KUKA KRL program: MyProgram_011().src

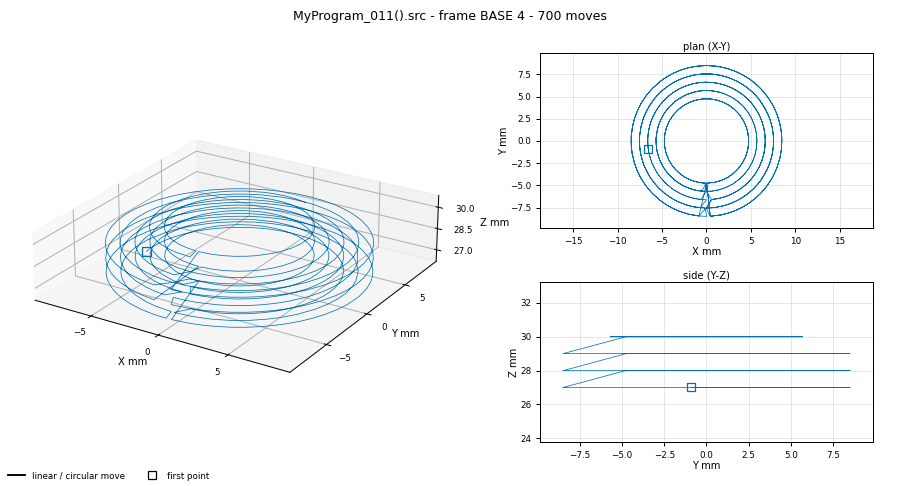
[picture p0: tool path of MyProgram_011().src in frame BASE 4, 700 of 700 moves have a stored position in this frame; points joined in program order, loops and branches not executed]
&ACCESS RVP
&REL 1
&PARAM TEMPLATE = C:\KRC\Roboter\Template\vorgabe
&PARAM EDITMASK = *
DEF MyProgram_011()
; ---- Setting reference (Base) ----
$BASE = BASE_DATA[4]

; --------------------------
; ---- Setting tool (TCP) ----
$TOOL = TOOL_DATA[3]
; --------------------------

$VEL.CP = VEL_APROX_PRINT
Startdeposition()
$VEL.CP = VEL_PRINT
LIN {X -6.5573,Y -0.8939,Z 27,A -3.0087,B 0,C 0,E1 0.1598,E2 90.0713} C_DIS
LIN {X -6.618,Y -0.1474,Z 27,A -2.9794,B 0,C 0,E1 0.1598,E2 90.0713} C_DIS
LIN {X -6.5928,Y 0.601,Z 27,A -2.9469,B 0,C 0,E1 0.1598,E2 90.0713} C_DIS
LIN {X -6.4833,Y 1.342,Z 27,A -2.9115,B 0,C 0,E1 0.1598,E2 90.0714} C_DIS
LIN {X -6.2883,Y 2.0652,Z 27,A -2.8738,B 0,C 0,E1 0.1598,E2 90.0714} C_DIS
LIN {X -6.0156,Y 2.7627,Z 27,A -2.8344,B 0,C 0,E1 0.1598,E2 90.0715} C_DIS
LIN {X -5.664,Y 3.4241,Z 27,A -2.7935,B 0,C 0,E1 0.1598,E2 90.0716} C_DIS
LIN {X -5.2401,Y 4.0414,Z 27,A -2.7519,B 0,C 0,E1 0.1598,E2 90.0717} C_DIS
LIN {X -4.7509,Y 4.6085,Z 27,A -2.7099,B 0,C 0,E1 0.1598,E2 90.0717} C_DIS
LIN {X -4.2004,Y 5.116,Z 27,A -2.6682,B 0,C 0,E1 0.1598,E2 90.0719} C_DIS
LIN {X -3.5961,Y 5.5584,Z 27,A -2.6273,B 0,C 0,E1 0.1598,E2 90.0719} C_DIS
LIN {X -2.9446,Y 5.9279,Z 27,A -2.5877,B 0,C 0,E1 0.1598,E2 90.0721} C_DIS
LIN {X -2.2557,Y 6.2218,Z 27,A -2.5499,B 0,C 0,E1 0.1598,E2 90.0721} C_DIS
LIN {X -1.5387,Y 6.4385,Z 27,A -2.5143,B 0,C 0,E1 0.1598,E2 90.0721} C_DIS
LIN {X -0.8014,Y 6.5698,Z 27,A -2.4815,B 0,C 0,E1 0.1598,E2 90.0723} C_DIS
LIN {X -0.0541,Y 6.618,Z 27,A -2.4519,B 0,C 0,E1 0.1598,E2 90.0723} C_DIS
LIN {X 0.6941,Y 6.5838,Z 27,A -2.4258,B 0,C 0,E1 0.1598,E2 90.0723} C_DIS
LIN {X 1.433,Y 6.4616,Z 27,A -2.4037,B 0,C 0,E1 0.1598,E2 90.0723} C_DIS
LIN {X 2.1541,Y 6.2595,Z 27,A -2.3856,B 0,C 0,E1 0.1598,E2 90.0723} C_DIS
LIN {X 2.8468,Y 5.9745,Z 27,A -2.3721,B 0,C 0,E1 0.1598,E2 90.0723} C_DIS
LIN {X 3.504,Y 5.6154,Z 27,A -2.3631,B 0,C 0,E1 0.1598,E2 90.0723} C_DIS
LIN {X 4.1162,Y 5.1839,Z 27,A -2.3588,B 0,C 0,E1 0.1598,E2 90.0723} C_DIS
LIN {X 4.6757,Y 4.6859,Z 27,A -2.3592,B 0,C 0,E1 0.1598,E2 90.0723} C_DIS
LIN {X 5.1746,Y 4.1272,Z 27,A -2.3645,B 0,C 0,E1 0.1598,E2 90.0723} C_DIS
LIN {X 5.6072,Y 3.5157,Z 27,A -2.3745,B 0,C 0,E1 0.1598,E2 90.0722} C_DIS
LIN {X 5.9685,Y 2.8598,Z 27,A -2.389,B 0,C 0,E1 0.1598,E2 90.0722} C_DIS
LIN {X 6.2523,Y 2.1668,Z 27,A -2.408,B 0,C 0,E1 0.1598,E2 90.0721} C_DIS
LIN {X 6.4581,Y 1.4468,Z 27,A -2.431,B 0,C 0,E1 0.1598,E2 90.0721} C_DIS
LIN {X 6.5825,Y 0.7083,Z 27,A -2.4579,B 0,C 0,E1 0.1598,E2 90.072} C_DIS
LIN {X 6.6179,Y -0.0399,Z 27,A -2.4884,B 0,C 0,E1 0.1598,E2 90.072} C_DIS
LIN {X 6.5713,Y -0.7872,Z 27,A -2.5219,B 0,C 0,E1 0.1598,E2 90.0719} C_DIS
LIN {X 6.4411,Y -1.5247,Z 27,A -2.5581,B 0,C 0,E1 0.1598,E2 90.0719} C_DIS
LIN {X 6.2271,Y -2.2424,Z 27,A -2.5965,B 0,C 0,E1 0.1598,E2 90.0719} C_DIS
LIN {X 5.9337,Y -2.9315,Z 27,A -2.6366,B 0,C 0,E1 0.1598,E2 90.0719} C_DIS
LIN {X 5.5647,Y -3.5833,Z 27,A -2.6779,B 0,C 0,E1 0.1598,E2 90.0718} C_DIS
LIN {X 5.1247,Y -4.1894,Z 27,A -2.7199,B 0,C 0,E1 0.1598,E2 90.0718} C_DIS
LIN {X 4.6171,Y -4.74,Z 27,A -2.762,B 0,C 0,E1 0.1598,E2 90.0718} C_DIS
LIN {X 4.0524,Y -5.2317,Z 27,A -2.8037,B 0,C 0,E1 0.1598,E2 90.0718} C_DIS
LIN {X 3.4359,Y -5.6569,Z 27,A -2.8444,B 0,C 0,E1 0.1598,E2 90.0717} C_DIS
LIN {X 2.7752,Y -6.0093,Z 27,A -2.8837,B 0,C 0,E1 0.1598,E2 90.0717} C_DIS
LIN {X 2.0782,Y -6.2831,Z 27,A -2.9209,B 0,C 0,E1 0.1598,E2 90.0717} C_DIS
LIN {X 1.3555,Y -6.4797,Z 27,A -2.9558,B 0,C 0,E1 0.1598,E2 90.0717} C_DIS
LIN {X 0.6148,Y -6.5905,Z 27,A -2.9877,B 0,C 0,E1 0.1598,E2 90.0716} C_DIS
LIN {X 0.6148,Y -6.5905,Z 27,A -2.9877,B 0,C 0,E1 0.1598,E2 90.0716} C_DIS
Enddeposition()
LIN {X 0.0294,Y -7.5563,Z 27,A -3.0492,B 0,C 0,E1 0.1598,E2 90.0703} C_DIS
Startdeposition()
$VEL.CP = VEL_PRINT
LIN {X 1.1276,Y -7.4726,Z 27,A -3.0064,B 0,C 0,E1 0.1598,E2 90.0715} C_DIS
LIN {X 2.4221,Y -7.16,Z 27,A -2.9457,B 0,C 0,E1 0.1598,E2 90.0716} C_DIS
LIN {X 3.4934,Y -6.6962,Z 27,A -2.8866,B 0,C 0,E1 0.1598,E2 90.0716} C_DIS
LIN {X 4.4261,Y -6.1265,Z 27,A -2.8281,B 0,C 0,E1 0.1598,E2 90.0716} C_DIS
LIN {X 5.3259,Y -5.356,Z 27,A -2.7622,B 0,C 0,E1 0.1598,E2 90.0716} C_DIS
LIN {X 5.8946,Y -4.7214,Z 27,A -2.7144,B 0,C 0,E1 0.1598,E2 90.0717} C_DIS
LIN {X 6.5048,Y -3.8483,Z 27,A -2.6545,B 0,C 0,E1 0.1598,E2 90.0716} C_DIS
LIN {X 7.0995,Y -2.5883,Z 27,A -2.5787,B 0,C 0,E1 0.1598,E2 90.0714} C_DIS
LIN {X 7.3873,Y -1.5916,Z 27,A -2.5259,B 0,C 0,E1 0.1598,E2 90.0716} C_DIS
LIN {X 7.5366,Y -0.5552,Z 27,A -2.4762,B 0,C 0,E1 0.1598,E2 90.0716} C_DIS
LIN {X 7.5438,Y 0.4481,Z 27,A -2.4333,B 0,C 0,E1 0.1598,E2 90.0717} C_DIS
LIN {X 7.425,Y 1.412,Z 27,A -2.3967,B 0,C 0,E1 0.1598,E2 90.0718} C_DIS
LIN {X 7.1966,Y 2.3052,Z 27,A -2.3672,B 0,C 0,E1 0.1598,E2 90.072} C_DIS
LIN {X 6.5668,Y 3.7404,Z 27,A -2.329,B 0,C 0,E1 0.1598,E2 90.0717} C_DIS
LIN {X 5.6905,Y 4.9679,Z 27,A -2.3091,B 0,C 0,E1 0.1598,E2 90.0717} C_DIS
LIN {X 5.2187,Y 5.4628,Z 27,A -2.3061,B 0,C 0,E1 0.1598,E2 90.0723} C_DIS
LIN {X 4.4003,Y 6.1444,Z 27,A -2.3073,B 0,C 0,E1 0.1598,E2 90.0723} C_DIS
LIN {X 3.4389,Y 6.7302,Z 27,A -2.3179,B 0,C 0,E1 0.1598,E2 90.0723} C_DIS
LIN {X 2.2888,Y 7.1954,Z 27,A -2.3408,B 0,C 0,E1 0.1598,E2 90.0723} C_DIS
LIN {X 1.4711,Y 7.4086,Z 27,A -2.362,B 0,C 0,E1 0.1598,E2 90.0723} C_DIS
LIN {X 0.6343,Y 7.527,Z 27,A -2.3879,B 0,C 0,E1 0.1598,E2 90.0723} C_DIS
LIN {X -0.2105,Y 7.5503,Z 27,A -2.4181,B 0,C 0,E1 0.1598,E2 90.0723} C_DIS
LIN {X -1.0526,Y 7.4788,Z 27,A -2.4522,B 0,C 0,E1 0.1598,E2 90.0723} C_DIS
LIN {X -2.0869,Y 7.2646,Z 27,A -2.4994,B 0,C 0,E1 0.1598,E2 90.0723} C_DIS
LIN {X -3.0794,Y 6.9019,Z 27,A -2.5514,B 0,C 0,E1 0.1598,E2 90.0721} C_DIS
LIN {X -4.0745,Y 6.365,Z 27,A -2.6107,B 0,C 0,E1 0.1598,E2 90.072} C_DIS
LIN {X -4.9827,Y 5.6816,Z 27,A -2.6729,B 0,C 0,E1 0.1598,E2 90.0718} C_DIS
LIN {X -5.5757,Y 5.0967,Z 27,A -2.7195,B 0,C 0,E1 0.1598,E2 90.0718} C_DIS
LIN {X -6.4393,Y 3.9543,Z 27,A -2.7989,B 0,C 0,E1 0.1598,E2 90.071} C_DIS
LIN {X -6.9322,Y 3.0073,Z 27,A -2.8574,B 0,C 0,E1 0.1598,E2 90.0713} C_DIS
LIN {X -7.1839,Y 2.346,Z 27,A -2.8948,B 0,C 0,E1 0.1598,E2 90.0715} C_DIS
LIN {X -7.5235,Y 0.721,Z 27,A -2.9747,B 0,C 0,E1 0.1598,E2 90.0703} C_DIS
LIN {X -7.5464,Y -0.4096,Z 27,A -3.0239,B 0,C 0,E1 0.1598,E2 90.0708} C_DIS
LIN {X -7.4299,Y -1.359,Z 27,A -3.06,B 0,C 0,E1 0.1598,E2 90.0711} C_DIS
LIN {X -7.2544,Y -2.1037,Z 27,A -3.0851,B 0,C 0,E1 0.1598,E2 90.0711} C_DIS
LIN {X -7.0048,Y -2.8269,Z 27,A -3.1065,B 0,C 0,E1 0.1598,E2 90.0711} C_DIS
LIN {X -6.5265,Y -3.8128,Z 27,A -3.1304,B 0,C 0,E1 0.1598,E2 90.0709} C_DIS
LIN {X -5.9309,Y -4.6747,Z 27,A -3.1451,B 0,C 0,E1 0.1598,E2 90.071} C_DIS
LIN {X -5.3766,Y -5.3032,Z 27,A -3.1515,B 0,C 0,E1 0.1598,E2 90.0712} C_DIS
LIN {X -4.7558,Y -5.8663,Z 27,A -3.1526,B 0,C 0,E1 0.1598,E2 90.0712} C_DIS
LIN {X -4.0775,Y -6.3584,Z 27,A -3.1486,B 0,C 0,E1 0.1598,E2 90.0712} C_DIS
LIN {X -3.3478,Y -6.7707,Z 27,A -3.1393,B 0,C 0,E1 0.1598,E2 90.0712} C_DIS
LIN {X -2.2931,Y -7.2004,Z 27,A -3.1188,B 0,C 0,E1 0.1598,E2 90.0713} C_DIS
LIN {X -1.43,Y -7.4212,Z 27,A -3.0966,B 0,C 0,E1 0.1598,E2 90.0714} C_DIS
LIN {X -0.2037,Y -7.5502,Z 27,A -3.0572,B 0,C 0,E1 0.1598,E2 90.0714} C_DIS
LIN {X -0.2037,Y -7.5502,Z 27,A -3.0572,B 0,C 0,E1 0.1598,E2 90.0714} C_DIS
Enddeposition()
LIN {X 0.0544,Y -8.4909,Z 27,A -3.0867,B 0,C 0,E1 0.1598,E2 90.0703} C_DIS
Startdeposition()
$VEL.CP = VEL_PRINT
LIN {X -0.8407,Y -8.4495,Z 27,A -3.1189,B 0,C 0,E1 0.1598,E2 90.0714} C_DIS
LIN {X -1.969,Y -8.2606,Z 27,A -3.1522,B 0,C 0,E1 0.1598,E2 90.0714} C_DIS
LIN {X -3.1017,Y -7.9005,Z 27,A -3.1784,B 0,C 0,E1 0.1598,E2 90.0712} C_DIS
LIN {X -3.874,Y -7.5517,Z 27,A -3.1919,B 0,C 0,E1 0.1598,E2 90.0712} C_DIS
LIN {X -4.6077,Y -7.1278,Z 27,A -3.2009,B 0,C 0,E1 0.1598,E2 90.0712} C_DIS
LIN {X -5.2957,Y -6.6329,Z 27,A -3.2051,B 0,C 0,E1 0.1598,E2 90.0712} C_DIS
LIN {X -6.1478,Y -5.8553,Z 27,A -3.2033,B 0,C 0,E1 0.1598,E2 90.071} C_DIS
LIN {X -6.812,Y -5.0692,Z 27,A -3.1944,B 0,C 0,E1 0.1598,E2 90.071} C_DIS
LIN {X -7.4625,Y -4.0464,Z 27,A -3.1748,B 0,C 0,E1 0.1598,E2 90.0708} C_DIS
LIN {X -7.8292,Y -3.2813,Z 27,A -3.1562,B 0,C 0,E1 0.1598,E2 90.071} C_DIS
LIN {X -8.1175,Y -2.4834,Z 27,A -3.133,B 0,C 0,E1 0.1598,E2 90.071} C_DIS
LIN {X -8.3794,Y -1.3682,Z 27,A -3.0953,B 0,C 0,E1 0.1598,E2 90.0709} C_DIS
LIN {X -8.4868,Y -0.2009,Z 27,A -3.0498,B 0,C 0,E1 0.1598,E2 90.0707} C_DIS
LIN {X -8.4719,Y 0.5615,Z 27,A -3.0174,B 0,C 0,E1 0.1598,E2 90.0711} C_DIS
LIN {X -8.2931,Y 1.8104,Z 27,A -2.9578,B 0,C 0,E1 0.1598,E2 90.0708} C_DIS
LIN {X -8.1092,Y 2.5151,Z 27,A -2.9218,B 0,C 0,E1 0.1598,E2 90.0713} C_DIS
LIN {X -7.7311,Y 3.502,Z 27,A -2.8661,B 0,C 0,E1 0.1598,E2 90.0713} C_DIS
LIN {X -7.3443,Y 4.2539,Z 27,A -2.8203,B 0,C 0,E1 0.1598,E2 90.0715} C_DIS
LIN {X -6.7611,Y 5.1353,Z 27,A -2.7615,B 0,C 0,E1 0.1598,E2 90.0715} C_DIS
LIN {X -6.0622,Y 5.9455,Z 27,A -2.7017,B 0,C 0,E1 0.1598,E2 90.0716} C_DIS
LIN {X -5.1243,Y 6.7675,Z 27,A -2.6324,B 0,C 0,E1 0.1598,E2 90.0717} C_DIS
LIN {X -4.4243,Y 7.245,Z 27,A -2.5866,B 0,C 0,E1 0.1598,E2 90.072} C_DIS
LIN {X -3.6802,Y 7.6502,Z 27,A -2.5421,B 0,C 0,E1 0.1598,E2 90.0721} C_DIS
LIN {X -2.8993,Y 7.9789,Z 27,A -2.4994,B 0,C 0,E1 0.1598,E2 90.0721} C_DIS
LIN {X -2.0894,Y 8.2279,Z 27,A -2.459,B 0,C 0,E1 0.1598,E2 90.0723} C_DIS
LIN {X -1.2587,Y 8.3946,Z 27,A -2.4213,B 0,C 0,E1 0.1598,E2 90.0723} C_DIS
LIN {X -0.0535,Y 8.4915,Z 27,A -2.3727,B 0,C 0,E1 0.1598,E2 90.0724} C_DIS
LIN {X 1.2628,Y 8.3964,Z 27,A -2.3281,B 0,C 0,E1 0.1598,E2 90.0724} C_DIS
LIN {X 2.4556,Y 8.1256,Z 27,A -2.2955,B 0,C 0,E1 0.1598,E2 90.0724} C_DIS
LIN {X 3.2184,Y 7.8542,Z 27,A -2.2788,B 0,C 0,E1 0.1598,E2 90.0724} C_DIS
LIN {X 3.9514,Y 7.5104,Z 27,A -2.2663,B 0,C 0,E1 0.1598,E2 90.0724} C_DIS
LIN {X 4.6492,Y 7.0998,Z 27,A -2.2579,B 0,C 0,E1 0.1598,E2 90.0724} C_DIS
LIN {X 5.3052,Y 6.6251,Z 27,A -2.2538,B 0,C 0,E1 0.1598,E2 90.0724} C_DIS
LIN {X 6.132,Y 5.8719,Z 27,A -2.2551,B 0,C 0,E1 0.1598,E2 90.0722} C_DIS
LIN {X 6.8769,Y 4.9736,Z 27,A -2.2656,B 0,C 0,E1 0.1598,E2 90.072} C_DIS
LIN {X 7.3469,Y 4.248,Z 27,A -2.2793,B 0,C 0,E1 0.1598,E2 90.0722} C_DIS
LIN {X 7.7408,Y 3.4783,Z 27,A -2.2975,B 0,C 0,E1 0.1598,E2 90.0722} C_DIS
LIN {X 8.0543,Y 2.6727,Z 27,A -2.3202,B 0,C 0,E1 0.1598,E2 90.0721} C_DIS
LIN {X 8.3335,Y 1.6286,Z 27,A -2.354,B 0,C 0,E1 0.1598,E2 90.0717} C_DIS
LIN {X 8.4815,Y 0.4189,Z 27,A -2.4,B 0,C 0,E1 0.1598,E2 90.0715} C_DIS
LIN {X 8.4392,Y -0.9319,Z 27,A -2.4589,B 0,C 0,E1 0.1598,E2 90.0714} C_DIS
LIN {X 8.2865,Y -1.8528,Z 27,A -2.5042,B 0,C 0,E1 0.1598,E2 90.0718} C_DIS
LIN {X 7.9336,Y -3.0156,Z 27,A -2.5665,B 0,C 0,E1 0.1598,E2 90.0714} C_DIS
LIN {X 7.5889,Y -3.7991,Z 27,A -2.6129,B 0,C 0,E1 0.1598,E2 90.0717} C_DIS
LIN {X 7.1674,Y -4.544,Z 27,A -2.6602,B 0,C 0,E1 0.1598,E2 90.0717} C_DIS
LIN {X 6.6729,Y -5.2426,Z 27,A -2.7081,B 0,C 0,E1 0.1598,E2 90.0717} C_DIS
LIN {X 6.1112,Y -5.8884,Z 27,A -2.7563,B 0,C 0,E1 0.1598,E2 90.0717} C_DIS
LIN {X 5.4874,Y -6.4744,Z 27,A -2.8041,B 0,C 0,E1 0.1598,E2 90.0717} C_DIS
LIN {X 4.8078,Y -6.9947,Z 27,A -2.8513,B 0,C 0,E1 0.1598,E2 90.0717} C_DIS
LIN {X 4.0792,Y -7.4439,Z 27,A -2.8971,B 0,C 0,E1 0.1598,E2 90.0717} C_DIS
LIN {X 3.3089,Y -7.8171,Z 27,A -2.9413,B 0,C 0,E1 0.1598,E2 90.0716} C_DIS
LIN {X 2.5048,Y -8.1107,Z 27,A -2.9833,B 0,C 0,E1 0.1598,E2 90.0716} C_DIS
LIN {X 1.6752,Y -8.3215,Z 27,A -3.0226,B 0,C 0,E1 0.1598,E2 90.0716} C_DIS
LIN {X 0.4289,Y -8.4809,Z 27,A -3.0751,B 0,C 0,E1 0.1598,E2 90.0715} C_DIS
LIN {X 0.4289,Y -8.4809,Z 27,A -3.0751,B 0,C 0,E1 0.1598,E2 90.0715} C_DIS
Enddeposition()
LIN {X 0.0007,Y -4.757,Z 28,A -2.9177,B 0,C 0,E1 0.1598,E2 90.0604} C_DIS
Startdeposition()
$VEL.CP = VEL_PRINT
LIN {X 0.0007,Y -4.757,Z 28,A -2.9234,B 0,C 0,E1 0.1598,E2 90.0661} C_DIS
LIN {X 0.963,Y -4.6517,Z 28,A -2.8885,B 0,C 0,E1 0.1598,E2 90.071} C_DIS
LIN {X 1.706,Y -4.4332,Z 28,A -2.8526,B 0,C 0,E1 0.1598,E2 90.0717} C_DIS
LIN {X 2.4029,Y -4.0959,Z 28,A -2.8127,B 0,C 0,E1 0.1598,E2 90.0717} C_DIS
LIN {X 3.0367,Y -3.6513,Z 28,A -2.7704,B 0,C 0,E1 0.1598,E2 90.0717} C_DIS
LIN {X 3.5915,Y -3.1111,Z 28,A -2.727,B 0,C 0,E1 0.1598,E2 90.0717} C_DIS
LIN {X 4.049,Y -2.4861,Z 28,A -2.6836,B 0,C 0,E1 0.1598,E2 90.0717} C_DIS
LIN {X 4.3992,Y -1.7952,Z 28,A -2.6413,B 0,C 0,E1 0.1598,E2 90.0717} C_DIS
LIN {X 4.6513,Y -0.9615,Z 28,A -2.5964,B 0,C 0,E1 0.1598,E2 90.0717} C_DIS
LIN {X 4.7407,Y -0.2897,Z 28,A -2.5647,B 0,C 0,E1 0.1598,E2 90.0719} C_DIS
LIN {X 4.7242,Y 0.4842,Z 28,A -2.5324,B 0,C 0,E1 0.1598,E2 90.0719} C_DIS
LIN {X 4.6298,Y 1.0574,Z 28,A -2.5116,B 0,C 0,E1 0.1598,E2 90.0719} C_DIS
LIN {X 4.3962,Y 1.7954,Z 28,A -2.4888,B 0,C 0,E1 0.1598,E2 90.0719} C_DIS
LIN {X 4.0466,Y 2.4862,Z 28,A -2.4723,B 0,C 0,E1 0.1598,E2 90.0719} C_DIS
LIN {X 3.5881,Y 3.1099,Z 28,A -2.4628,B 0,C 0,E1 0.1598,E2 90.0721} C_DIS
LIN {X 3.0356,Y 3.6523,Z 28,A -2.4602,B 0,C 0,E1 0.1598,E2 90.0721} C_DIS
LIN {X 2.4016,Y 4.0966,Z 28,A -2.4647,B 0,C 0,E1 0.1598,E2 90.0721} C_DIS
LIN {X 1.8838,Y 4.3598,Z 28,A -2.4727,B 0,C 0,E1 0.1598,E2 90.0722} C_DIS
LIN {X 1.1502,Y 4.6074,Z 28,A -2.4893,B 0,C 0,E1 0.1598,E2 90.0722} C_DIS
LIN {X 0.3864,Y 4.7336,Z 28,A -2.5121,B 0,C 0,E1 0.1598,E2 90.0722} C_DIS
LIN {X -0.3879,Y 4.7339,Z 28,A -2.5407,B 0,C 0,E1 0.1598,E2 90.0722} C_DIS
LIN {X -1.1516,Y 4.607,Z 28,A -2.5742,B 0,C 0,E1 0.1598,E2 90.0722} C_DIS
LIN {X -1.8851,Y 4.3592,Z 28,A -2.6117,B 0,C 0,E1 0.1598,E2 90.0721} C_DIS
LIN {X -2.5682,Y 3.9948,Z 28,A -2.6522,B 0,C 0,E1 0.1598,E2 90.072} C_DIS
LIN {X -3.1841,Y 3.5255,Z 28,A -2.6947,B 0,C 0,E1 0.1598,E2 90.0719} C_DIS
LIN {X -3.7154,Y 2.9617,Z 28,A -2.7381,B 0,C 0,E1 0.1598,E2 90.0718} C_DIS
LIN {X -4.1464,Y 2.3182,Z 28,A -2.7811,B 0,C 0,E1 0.1598,E2 90.0717} C_DIS
LIN {X -4.4674,Y 1.6136,Z 28,A -2.8227,B 0,C 0,E1 0.1598,E2 90.0716} C_DIS
LIN {X -4.6724,Y 0.8667,Z 28,A -2.8617,B 0,C 0,E1 0.1598,E2 90.0715} C_DIS
LIN {X -4.7506,Y 0.0961,Z 28,A -2.8972,B 0,C 0,E1 0.1598,E2 90.0714} C_DIS
LIN {X -4.7017,Y -0.6768,Z 28,A -2.928,B 0,C 0,E1 0.1598,E2 90.0714} C_DIS
LIN {X -4.5299,Y -1.4319,Z 28,A -2.9537,B 0,C 0,E1 0.1598,E2 90.0714} C_DIS
LIN {X -4.2369,Y -2.1487,Z 28,A -2.9733,B 0,C 0,E1 0.1598,E2 90.0714} C_DIS
LIN {X -3.8305,Y -2.8078,Z 28,A -2.9863,B 0,C 0,E1 0.1598,E2 90.0714} C_DIS
LIN {X -3.323,Y -3.3926,Z 28,A -2.9924,B 0,C 0,E1 0.1598,E2 90.0714} C_DIS
LIN {X -2.7279,Y -3.8877,Z 28,A -2.9916,B 0,C 0,E1 0.1598,E2 90.0714} C_DIS
LIN {X -2.0599,Y -4.2793,Z 28,A -2.9837,B 0,C 0,E1 0.1598,E2 90.0715} C_DIS
LIN {X -1.3374,Y -4.5575,Z 28,A -2.969,B 0,C 0,E1 0.1598,E2 90.0715} C_DIS
LIN {X -0.5793,Y -4.7151,Z 28,A -2.9479,B 0,C 0,E1 0.1598,E2 90.0716} C_DIS
LIN {X 0.0007,Y -4.757,Z 28,A -2.9284,B 0,C 0,E1 0.1598,E2 90.0716} C_DIS
Enddeposition()
LIN {X 0.0007,Y -4.757,Z 28,A -2.9284,B 0,C 0,E1 0.1598,E2 90.0716} C_DIS
Startdeposition()
$VEL.CP = VEL_PRINT
LIN {X -0.5455,Y -5.6575,Z 28,A -2.9862,B 0,C 0,E1 0.1598,E2 90.071} C_DIS
LIN {X -1.4457,Y -5.5027,Z 28,A -3.0132,B 0,C 0,E1 0.1598,E2 90.0715} C_DIS
LIN {X -2.5876,Y -5.0681,Z 28,A -3.0366,B 0,C 0,E1 0.1598,E2 90.0714} C_DIS
LIN {X -3.4004,Y -4.5542,Z 28,A -3.0447,B 0,C 0,E1 0.1598,E2 90.0714} C_DIS
LIN {X -3.9832,Y -4.0522,Z 28,A -3.0447,B 0,C 0,E1 0.1598,E2 90.0714} C_DIS
LIN {X -4.4942,Y -3.4775,Z 28,A -3.0392,B 0,C 0,E1 0.1598,E2 90.0714} C_DIS
LIN {X -4.9245,Y -2.8399,Z 28,A -3.028,B 0,C 0,E1 0.1598,E2 90.0714} C_DIS
LIN {X -5.2643,Y -2.1496,Z 28,A -3.0112,B 0,C 0,E1 0.1598,E2 90.0714} C_DIS
LIN {X -5.5044,Y -1.4186,Z 28,A -2.9891,B 0,C 0,E1 0.1598,E2 90.0714} C_DIS
LIN {X -5.6444,Y -0.6623,Z 28,A -2.9623,B 0,C 0,E1 0.1598,E2 90.0714} C_DIS
LIN {X -5.6825,Y 0.2984,Z 28,A -2.9228,B 0,C 0,E1 0.1598,E2 90.0711} C_DIS
LIN {X -5.4173,Y 1.7389,Z 28,A -2.8517,B 0,C 0,E1 0.1598,E2 90.0707} C_DIS
LIN {X -5.052,Y 2.6035,Z 28,A -2.8023,B 0,C 0,E1 0.1598,E2 90.0714} C_DIS
LIN {X -4.6641,Y 3.2461,Z 28,A -2.7611,B 0,C 0,E1 0.1598,E2 90.0717} C_DIS
LIN {X -4.1969,Y 3.8336,Z 28,A -2.7191,B 0,C 0,E1 0.1598,E2 90.0717} C_DIS
LIN {X -3.5124,Y 4.4758,Z 28,A -2.6667,B 0,C 0,E1 0.1598,E2 90.0717} C_DIS
LIN {X -2.2637,Y 5.2198,Z 28,A -2.5891,B 0,C 0,E1 0.1598,E2 90.0719} C_DIS
LIN {X -0.7561,Y 5.64,Z 28,A -2.5159,B 0,C 0,E1 0.1598,E2 90.0721} C_DIS
LIN {X 0.399,Y 5.6757,Z 28,A -2.4719,B 0,C 0,E1 0.1598,E2 90.0723} C_DIS
LIN {X 1.5931,Y 5.463,Z 28,A -2.4368,B 0,C 0,E1 0.1598,E2 90.0723} C_DIS
LIN {X 2.1802,Y 5.2494,Z 28,A -2.4242,B 0,C 0,E1 0.1598,E2 90.0723} C_DIS
LIN {X 2.9234,Y 4.8747,Z 28,A -2.4127,B 0,C 0,E1 0.1598,E2 90.0723} C_DIS
LIN {X 3.6043,Y 4.396,Z 28,A -2.4078,B 0,C 0,E1 0.1598,E2 90.0723} C_DIS
LIN {X 4.2072,Y 3.8224,Z 28,A -2.4099,B 0,C 0,E1 0.1598,E2 90.0722} C_DIS
LIN {X 4.7201,Y 3.167,Z 28,A -2.4188,B 0,C 0,E1 0.1598,E2 90.0721} C_DIS
LIN {X 5.1314,Y 2.4435,Z 28,A -2.4343,B 0,C 0,E1 0.1598,E2 90.0721} C_DIS
LIN {X 5.4343,Y 1.6684,Z 28,A -2.456,B 0,C 0,E1 0.1598,E2 90.0719} C_DIS
LIN {X 5.6202,Y 0.8572,Z 28,A -2.4837,B 0,C 0,E1 0.1598,E2 90.0719} C_DIS
LIN {X 5.6861,Y 0.0275,Z 28,A -2.5165,B 0,C 0,E1 0.1598,E2 90.0719} C_DIS
LIN {X 5.6288,Y -0.803,Z 28,A -2.5539,B 0,C 0,E1 0.1598,E2 90.0718} C_DIS
LIN {X 5.4504,Y -1.616,Z 28,A -2.5951,B 0,C 0,E1 0.1598,E2 90.0718} C_DIS
LIN {X 5.1549,Y -2.394,Z 28,A -2.6391,B 0,C 0,E1 0.1598,E2 90.0718} C_DIS
LIN {X 4.7488,Y -3.1201,Z 28,A -2.6849,B 0,C 0,E1 0.1598,E2 90.0718} C_DIS
LIN {X 4.242,Y -3.7799,Z 28,A -2.7317,B 0,C 0,E1 0.1598,E2 90.0718} C_DIS
LIN {X 3.645,Y -4.3593,Z 28,A -2.7783,B 0,C 0,E1 0.1598,E2 90.0718} C_DIS
LIN {X 2.9696,Y -4.845,Z 28,A -2.8238,B 0,C 0,E1 0.1598,E2 90.0717} C_DIS
LIN {X 2.2302,Y -5.2264,Z 28,A -2.8672,B 0,C 0,E1 0.1598,E2 90.0717} C_DIS
LIN {X 1.4431,Y -5.4959,Z 28,A -2.9075,B 0,C 0,E1 0.1598,E2 90.0717} C_DIS
LIN {X 0.6252,Y -5.648,Z 28,A -2.944,B 0,C 0,E1 0.1598,E2 90.0717} C_DIS
LIN {X 0.002,Y -5.6862,Z 28,A -2.9685,B 0,C 0,E1 0.1598,E2 90.0717} C_DIS
Enddeposition()
LIN {X 0.002,Y -5.6862,Z 28,A -2.9685,B 0,C 0,E1 0.1598,E2 90.0717} C_DIS
Startdeposition()
$VEL.CP = VEL_PRINT
LIN {X 0.5678,Y -6.5933,Z 28,A -2.9859,B 0,C 0,E1 0.1598,E2 90.071} C_DIS
LIN {X 1.325,Y -6.4863,Z 28,A -2.9541,B 0,C 0,E1 0.1598,E2 90.0716} C_DIS
LIN {X 2.0641,Y -6.2903,Z 28,A -2.9187,B 0,C 0,E1 0.1598,E2 90.0716} C_DIS
LIN {X 2.7755,Y -6.0094,Z 28,A -2.8806,B 0,C 0,E1 0.1598,E2 90.0716} C_DIS
LIN {X 3.4496,Y -5.6484,Z 28,A -2.8405,B 0,C 0,E1 0.1598,E2 90.0717} C_DIS
LIN {X 4.0795,Y -5.2147,Z 28,A -2.7989,B 0,C 0,E1 0.1598,E2 90.0717} C_DIS
LIN {X 4.653,Y -4.7087,Z 28,A -2.7563,B 0,C 0,E1 0.1598,E2 90.0717} C_DIS
LIN {X 5.1645,Y -4.1402,Z 28,A -2.7133,B 0,C 0,E1 0.1598,E2 90.0717} C_DIS
LIN {X 5.6083,Y -3.5172,Z 28,A -2.6704,B 0,C 0,E1 0.1598,E2 90.0718} C_DIS
LIN {X 5.9776,Y -2.8477,Z 28,A -2.6283,B 0,C 0,E1 0.1598,E2 90.0718} C_DIS
LIN {X 6.2652,Y -2.1391,Z 28,A -2.5875,B 0,C 0,E1 0.1598,E2 90.0718} C_DIS
LIN {X 6.4688,Y -1.4022,Z 28,A -2.5487,B 0,C 0,E1 0.1598,E2 90.0718} C_DIS
LIN {X 6.5866,Y -0.6466,Z 28,A -2.5122,B 0,C 0,E1 0.1598,E2 90.0719} C_DIS
LIN {X 6.6167,Y 0.1172,Z 28,A -2.4785,B 0,C 0,E1 0.1598,E2 90.0719} C_DIS
LIN {X 6.5616,Y 0.88,Z 28,A -2.4481,B 0,C 0,E1 0.1598,E2 90.0719} C_DIS
LIN {X 6.4145,Y 1.6304,Z 28,A -2.4216,B 0,C 0,E1 0.1598,E2 90.072} C_DIS
LIN {X 6.1829,Y 2.3591,Z 28,A -2.3991,B 0,C 0,E1 0.1598,E2 90.072} C_DIS
LIN {X 5.8718,Y 3.0575,Z 28,A -2.3809,B 0,C 0,E1 0.1598,E2 90.0721} C_DIS
LIN {X 5.4808,Y 3.7146,Z 28,A -2.3674,B 0,C 0,E1 0.1598,E2 90.0721} C_DIS
LIN {X 5.0165,Y 4.3223,Z 28,A -2.3588,B 0,C 0,E1 0.1598,E2 90.0722} C_DIS
LIN {X 4.4832,Y 4.8704,Z 28,A -2.3552,B 0,C 0,E1 0.1598,E2 90.0722} C_DIS
LIN {X 3.8915,Y 5.355,Z 28,A -2.3565,B 0,C 0,E1 0.1598,E2 90.0722} C_DIS
LIN {X 2.9648,Y 5.9228,Z 28,A -2.3665,B 0,C 0,E1 0.1598,E2 90.0722} C_DIS
LIN {X 2.0894,Y 6.2821,Z 28,A -2.3837,B 0,C 0,E1 0.1598,E2 90.0723} C_DIS
LIN {X 1.3578,Y 6.4765,Z 28,A -2.4025,B 0,C 0,E1 0.1598,E2 90.0723} C_DIS
LIN {X 0.6094,Y 6.5902,Z 28,A -2.4253,B 0,C 0,E1 0.1598,E2 90.0723} C_DIS
LIN {X -0.1472,Y 6.6173,Z 28,A -2.4521,B 0,C 0,E1 0.1598,E2 90.0723} C_DIS
LIN {X -0.902,Y 6.5575,Z 28,A -2.4825,B 0,C 0,E1 0.1598,E2 90.0723} C_DIS
LIN {X -1.6446,Y 6.4101,Z 28,A -2.5161,B 0,C 0,E1 0.1598,E2 90.0723} C_DIS
LIN {X -2.3661,Y 6.1808,Z 28,A -2.5524,B 0,C 0,E1 0.1598,E2 90.0721} C_DIS
LIN {X -3.0561,Y 5.8694,Z 28,A -2.591,B 0,C 0,E1 0.1598,E2 90.0721} C_DIS
LIN {X -3.7083,Y 5.485,Z 28,A -2.6313,B 0,C 0,E1 0.1598,E2 90.072} C_DIS
LIN {X -4.31,Y 5.0253,Z 28,A -2.6728,B 0,C 0,E1 0.1598,E2 90.072} C_DIS
LIN {X -4.8551,Y 4.4999,Z 28,A -2.7151,B 0,C 0,E1 0.1598,E2 90.0718} C_DIS
LIN {X -5.3367,Y 3.9155,Z 28,A -2.7575,B 0,C 0,E1 0.1598,E2 90.0718} C_DIS
LIN {X -5.7495,Y 3.2807,Z 28,A -2.7995,B 0,C 0,E1 0.1598,E2 90.0716} C_DIS
LIN {X -6.0883,Y 2.6037,Z 28,A -2.8405,B 0,C 0,E1 0.1598,E2 90.0716} C_DIS
LIN {X -6.3434,Y 1.8907,Z 28,A -2.88,B 0,C 0,E1 0.1598,E2 90.0715} C_DIS
LIN {X -6.5164,Y 1.1537,Z 28,A -2.9174,B 0,C 0,E1 0.1598,E2 90.0715} C_DIS
LIN {X -6.6071,Y 0.4021,Z 28,A -2.9525,B 0,C 0,E1 0.1598,E2 90.0713} C_DIS
LIN {X -6.6087,Y -0.3549,Z 28,A -2.9845,B 0,C 0,E1 0.1598,E2 90.0713} C_DIS
LIN {X -6.528,Y -1.1077,Z 28,A -3.0133,B 0,C 0,E1 0.1598,E2 90.0713} C_DIS
LIN {X -6.358,Y -1.8455,Z 28,A -3.0383,B 0,C 0,E1 0.1598,E2 90.0713} C_DIS
LIN {X -6.1068,Y -2.5598,Z 28,A -3.0593,B 0,C 0,E1 0.1598,E2 90.0713} C_DIS
LIN {X -5.7739,Y -3.2398,Z 28,A -3.0758,B 0,C 0,E1 0.1598,E2 90.0713} C_DIS
LIN {X -5.3655,Y -3.8775,Z 28,A -3.0878,B 0,C 0,E1 0.1598,E2 90.0713} C_DIS
LIN {X -4.8869,Y -4.4644,Z 28,A -3.0951,B 0,C 0,E1 0.1598,E2 90.0713} C_DIS
LIN {X -4.3445,Y -4.9926,Z 28,A -3.0976,B 0,C 0,E1 0.1598,E2 90.0713} C_DIS
LIN {X -3.7454,Y -5.4555,Z 28,A -3.0952,B 0,C 0,E1 0.1598,E2 90.0713} C_DIS
LIN {X -3.0991,Y -5.8496,Z 28,A -3.0882,B 0,C 0,E1 0.1598,E2 90.0713} C_DIS
LIN {X -2.4107,Y -6.1652,Z 28,A -3.0764,B 0,C 0,E1 0.1598,E2 90.0714} C_DIS
LIN {X -1.6904,Y -6.3984,Z 28,A -3.0599,B 0,C 0,E1 0.1598,E2 90.0714} C_DIS
LIN {X -0.9489,Y -6.5516,Z 28,A -3.0392,B 0,C 0,E1 0.1598,E2 90.0715} C_DIS
LIN {X -0.0052,Y -6.6206,Z 28,A -3.0075,B 0,C 0,E1 0.1598,E2 90.0715} C_DIS
Enddeposition()
LIN {X -0.0052,Y -6.6206,Z 28,A -3.0075,B 0,C 0,E1 0.1598,E2 90.0715} C_DIS
Startdeposition()
$VEL.CP = VEL_PRINT
LIN {X -0.6833,Y -7.5227,Z 28,A -3.0703,B 0,C 0,E1 0.1598,E2 90.0709} C_DIS
LIN {X -1.43,Y -7.4212,Z 28,A -3.0939,B 0,C 0,E1 0.1598,E2 90.0714} C_DIS
LIN {X -2.2913,Y -7.201,Z 28,A -3.1162,B 0,C 0,E1 0.1598,E2 90.0714} C_DIS
LIN {X -3.3368,Y -6.7761,Z 28,A -3.1364,B 0,C 0,E1 0.1598,E2 90.0713} C_DIS
LIN {X -4.0516,Y -6.3742,Z 28,A -3.1456,B 0,C 0,E1 0.1598,E2 90.0713} C_DIS
LIN {X -4.7187,Y -5.8976,Z 28,A -3.1499,B 0,C 0,E1 0.1598,E2 90.0713} C_DIS
LIN {X -5.3306,Y -5.3517,Z 28,A -3.1492,B 0,C 0,E1 0.1598,E2 90.0713} C_DIS
LIN {X -5.8794,Y -4.7423,Z 28,A -3.1435,B 0,C 0,E1 0.1598,E2 90.0712} C_DIS
LIN {X -6.3583,Y -4.0767,Z 28,A -3.1329,B 0,C 0,E1 0.1598,E2 90.0712} C_DIS
LIN {X -6.7613,Y -3.3628,Z 28,A -3.1174,B 0,C 0,E1 0.1598,E2 90.0712} C_DIS
LIN {X -7.0887,Y -2.611,Z 28,A -3.0977,B 0,C 0,E1 0.1598,E2 90.0712} C_DIS
LIN {X -7.3295,Y -1.8272,Z 28,A -3.0734,B 0,C 0,E1 0.1598,E2 90.0712} C_DIS
LIN {X -7.484,Y -1.0219,Z 28,A -3.045,B 0,C 0,E1 0.1598,E2 90.0712} C_DIS
LIN {X -7.5549,Y 0.1757,Z 28,A -2.9967,B 0,C 0,E1 0.1598,E2 90.0709} C_DIS
LIN {X -7.3952,Y 1.5541,Z 28,A -2.9322,B 0,C 0,E1 0.1598,E2 90.0705} C_DIS
LIN {X -7.1329,Y 2.4973,Z 28,A -2.8834,B 0,C 0,E1 0.1598,E2 90.0712} C_DIS
LIN {X -6.7699,Y 3.3575,Z 28,A -2.8338,B 0,C 0,E1 0.1598,E2 90.0714} C_DIS
LIN {X -5.9032,Y 4.7191,Z 28,A -2.7438,B 0,C 0,E1 0.1598,E2 90.0709} C_DIS
LIN {X -5.2951,Y 5.3855,Z 28,A -2.694,B 0,C 0,E1 0.1598,E2 90.0717} C_DIS
LIN {X -4.757,Y 5.8666,Z 28,A -2.6539,B 0,C 0,E1 0.1598,E2 90.0719} C_DIS
LIN {X -4.1759,Y 6.2949,Z 28,A -2.6145,B 0,C 0,E1 0.1598,E2 90.0719} C_DIS
LIN {X -3.5561,Y 6.665,Z 28,A -2.576,B 0,C 0,E1 0.1598,E2 90.0721} C_DIS
LIN {X -2.5752,Y 7.1043,Z 28,A -2.5212,B 0,C 0,E1 0.1598,E2 90.0721} C_DIS
LIN {X -1.4796,Y 7.407,Z 28,A -2.468,B 0,C 0,E1 0.1598,E2 90.0722} C_DIS
LIN {X -0.4661,Y 7.5426,Z 28,A -2.4249,B 0,C 0,E1 0.1598,E2 90.0723} C_DIS
LIN {X 0.7661,Y 7.5148,Z 28,A -2.3806,B 0,C 0,E1 0.1598,E2 90.0723} C_DIS
LIN {X 1.6891,Y 7.3611,Z 28,A -2.353,B 0,C 0,E1 0.1598,E2 90.0724} C_DIS
LIN {X 2.8073,Y 7.0176,Z 28,A -2.3262,B 0,C 0,E1 0.1598,E2 90.0724} C_DIS
LIN {X 4.0105,Y 6.4045,Z 28,A -2.3077,B 0,C 0,E1 0.1598,E2 90.0722} C_DIS
LIN {X 4.8373,Y 5.806,Z 28,A -2.3026,B 0,C 0,E1 0.1598,E2 90.0722} C_DIS
LIN {X 5.4597,Y 5.2216,Z 28,A -2.3045,B 0,C 0,E1 0.1598,E2 90.0723} C_DIS
LIN {X 6.0154,Y 4.5735,Z 28,A -2.3114,B 0,C 0,E1 0.1598,E2 90.0722} C_DIS
LIN {X 7.0188,Y 2.8045,Z 28,A -2.349,B 0,C 0,E1 0.1598,E2 90.0715} C_DIS
LIN {X 7.3743,Y 1.6355,Z 28,A -2.3857,B 0,C 0,E1 0.1598,E2 90.0715} C_DIS
LIN {X 7.504,Y 0.8928,Z 28,A -2.4129,B 0,C 0,E1 0.1598,E2 90.0719} C_DIS
LIN {X 7.5568,Y -0.0903,Z 28,A -2.4527,B 0,C 0,E1 0.1598,E2 90.0717} C_DIS
LIN {X 7.4782,Y -1.0928,Z 28,A -2.4983,B 0,C 0,E1 0.1598,E2 90.0717} C_DIS
LIN {X 7.2547,Y -2.1035,Z 28,A -2.5496,B 0,C 0,E1 0.1598,E2 90.0717} C_DIS
LIN {X 6.8881,Y -3.1065,Z 28,A -2.6057,B 0,C 0,E1 0.1598,E2 90.0715} C_DIS
LIN {X 6.17,Y -4.3555,Z 28,A -2.6851,B 0,C 0,E1 0.1598,E2 90.0713} C_DIS
LIN {X 5.6687,Y -4.9892,Z 28,A -2.731,B 0,C 0,E1 0.1598,E2 90.0717} C_DIS
LIN {X 5.1048,Y -5.5679,Z 28,A -2.7764,B 0,C 0,E1 0.1598,E2 90.0717} C_DIS
LIN {X 4.4805,Y -6.081,Z 28,A -2.8212,B 0,C 0,E1 0.1598,E2 90.0717} C_DIS
LIN {X 3.8048,Y -6.524,Z 28,A -2.8648,B 0,C 0,E1 0.1598,E2 90.0717} C_DIS
LIN {X 2.9021,Y -6.9773,Z 28,A -2.9172,B 0,C 0,E1 0.1598,E2 90.0716} C_DIS
LIN {X 1.6187,Y -7.3816,Z 28,A -2.9815,B 0,C 0,E1 0.1598,E2 90.0716} C_DIS
LIN {X 0.5862,Y -7.5345,Z 28,A -3.0259,B 0,C 0,E1 0.1598,E2 90.0716} C_DIS
LIN {X -0.0287,Y -7.5545,Z 28,A -3.0493,B 0,C 0,E1 0.1598,E2 90.0716} C_DIS
Enddeposition()
LIN {X -0.0287,Y -7.5545,Z 28,A -3.0493,B 0,C 0,E1 0.1598,E2 90.0716} C_DIS
Startdeposition()
$VEL.CP = VEL_PRINT
LIN {X 0.4292,Y -8.4808,Z 28,A -3.0715,B 0,C 0,E1 0.1598,E2 90.0709} C_DIS
LIN {X 1.6611,Y -8.3244,Z 28,A -3.0202,B 0,C 0,E1 0.1598,E2 90.0715} C_DIS
LIN {X 2.4827,Y -8.1178,Z 28,A -2.9814,B 0,C 0,E1 0.1598,E2 90.0715} C_DIS
LIN {X 3.2792,Y -7.8295,Z 28,A -2.9399,B 0,C 0,E1 0.1598,E2 90.0716} C_DIS
LIN {X 4.0434,Y -7.4642,Z 28,A -2.8963,B 0,C 0,E1 0.1598,E2 90.0716} C_DIS
LIN {X 4.767,Y -7.0237,Z 28,A -2.851,B 0,C 0,E1 0.1598,E2 90.0716} C_DIS
LIN {X 5.4431,Y -6.5133,Z 28,A -2.8044,B 0,C 0,E1 0.1598,E2 90.0717} C_DIS
LIN {X 6.0649,Y -5.938,Z 28,A -2.7571,B 0,C 0,E1 0.1598,E2 90.0717} C_DIS
LIN {X 6.6264,Y -5.3037,Z 28,A -2.7094,B 0,C 0,E1 0.1598,E2 90.0717} C_DIS
LIN {X 7.2913,Y -4.3515,Z 28,A -2.6442,B 0,C 0,E1 0.1598,E2 90.0717} C_DIS
LIN {X 7.8505,Y -3.2273,Z 28,A -2.5755,B 0,C 0,E1 0.1598,E2 90.0714} C_DIS
LIN {X 8.2285,Y -2.0926,Z 28,A -2.5132,B 0,C 0,E1 0.1598,E2 90.0715} C_DIS
LIN {X 8.4282,Y -1.0288,Z 28,A -2.4606,B 0,C 0,E1 0.1598,E2 90.0716} C_DIS
LIN {X 8.4916,Y 0.0464,Z 28,A -2.4124,B 0,C 0,E1 0.1598,E2 90.0716} C_DIS
LIN {X 8.4286,Y 1.0254,Z 28,A -2.3732,B 0,C 0,E1 0.1598,E2 90.0719} C_DIS
LIN {X 8.2241,Y 2.1097,Z 28,A -2.3344,B 0,C 0,E1 0.1598,E2 90.0719} C_DIS
LIN {X 7.892,Y 3.1225,Z 28,A -2.3036,B 0,C 0,E1 0.1598,E2 90.0719} C_DIS
LIN {X 7.5388,Y 3.8987,Z 28,A -2.2838,B 0,C 0,E1 0.1598,E2 90.0722} C_DIS
LIN {X 7.1096,Y 4.6355,Z 28,A -2.2683,B 0,C 0,E1 0.1598,E2 90.0722} C_DIS
LIN {X 6.4165,Y 5.5598,Z 28,A -2.2545,B 0,C 0,E1 0.1598,E2 90.0721} C_DIS
LIN {X 5.6064,Y 6.3725,Z 28,A -2.2499,B 0,C 0,E1 0.1598,E2 90.0721} C_DIS
LIN {X 4.9393,Y 6.902,Z 28,A -2.2522,B 0,C 0,E1 0.1598,E2 90.0724} C_DIS
LIN {X 4.2222,Y 7.3614,Z 28,A -2.2593,B 0,C 0,E1 0.1598,E2 90.0724} C_DIS
LIN {X 3.4632,Y 7.7476,Z 28,A -2.2709,B 0,C 0,E1 0.1598,E2 90.0724} C_DIS
LIN {X 2.6693,Y 8.0561,Z 28,A -2.2872,B 0,C 0,E1 0.1598,E2 90.0724} C_DIS
LIN {X 1.8485,Y 8.2832,Z 28,A -2.3079,B 0,C 0,E1 0.1598,E2 90.0724} C_DIS
LIN {X 1.0091,Y 8.4272,Z 28,A -2.3328,B 0,C 0,E1 0.1598,E2 90.0724} C_DIS
LIN {X -0.0535,Y 8.4915,Z 28,A -2.3694,B 0,C 0,E1 0.1598,E2 90.0724} C_DIS
LIN {X -1.2512,Y 8.3956,Z 28,A -2.4176,B 0,C 0,E1 0.1598,E2 90.0724} C_DIS
LIN {X -2.0826,Y 8.2295,Z 28,A -2.4554,B 0,C 0,E1 0.1598,E2 90.0723} C_DIS
LIN {X -2.8932,Y 7.981,Z 28,A -2.4958,B 0,C 0,E1 0.1598,E2 90.0723} C_DIS
LIN {X -3.6748,Y 7.6527,Z 28,A -2.5385,B 0,C 0,E1 0.1598,E2 90.0721} C_DIS
LIN {X -4.4197,Y 7.2478,Z 28,A -2.583,B 0,C 0,E1 0.1598,E2 90.0721} C_DIS
LIN {X -5.1203,Y 6.7704,Z 28,A -2.629,B 0,C 0,E1 0.1598,E2 90.072} C_DIS
LIN {X -6.0622,Y 5.9455,Z 28,A -2.6983,B 0,C 0,E1 0.1598,E2 90.0716} C_DIS
LIN {X -6.759,Y 5.138,Z 28,A -2.7581,B 0,C 0,E1 0.1598,E2 90.0716} C_DIS
LIN {X -7.3429,Y 4.2563,Z 28,A -2.8168,B 0,C 0,E1 0.1598,E2 90.0715} C_DIS
LIN {X -7.7302,Y 3.5041,Z 28,A -2.8628,B 0,C 0,E1 0.1598,E2 90.0715} C_DIS
LIN {X -8.1087,Y 2.5166,Z 28,A -2.9181,B 0,C 0,E1 0.1598,E2 90.0711} C_DIS
LIN {X -8.3768,Y 1.3752,Z 28,A -2.976,B 0,C 0,E1 0.1598,E2 90.0709} C_DIS
LIN {X -8.4719,Y 0.5625,Z 28,A -3.0139,B 0,C 0,E1 0.1598,E2 90.071} C_DIS
LIN {X -8.4654,Y -0.6204,Z 28,A -3.0633,B 0,C 0,E1 0.1598,E2 90.0707} C_DIS
LIN {X -8.3785,Y -1.3738,Z 28,A -3.0923,B 0,C 0,E1 0.1598,E2 90.071} C_DIS
LIN {X -8.1326,Y -2.4291,Z 28,A -3.1277,B 0,C 0,E1 0.1598,E2 90.0709} C_DIS
LIN {X -7.843,Y -3.2461,Z 28,A -3.1518,B 0,C 0,E1 0.1598,E2 90.071} C_DIS
LIN {X -7.4713,Y -4.0292,Z 28,A -3.1712,B 0,C 0,E1 0.1598,E2 90.071} C_DIS
LIN {X -6.8125,Y -5.0685,Z 28,A -3.1908,B 0,C 0,E1 0.1598,E2 90.0708} C_DIS
LIN {X -6.2115,Y -5.7883,Z 28,A -3.1994,B 0,C 0,E1 0.1598,E2 90.071} C_DIS
LIN {X -5.2984,Y -6.6307,Z 28,A -3.2015,B 0,C 0,E1 0.1598,E2 90.071} C_DIS
LIN {X -4.6103,Y -7.1261,Z 28,A -3.1974,B 0,C 0,E1 0.1598,E2 90.0712} C_DIS
LIN {X -3.8762,Y -7.5505,Z 28,A -3.1885,B 0,C 0,E1 0.1598,E2 90.0712} C_DIS
LIN {X -3.1035,Y -7.8997,Z 28,A -3.1751,B 0,C 0,E1 0.1598,E2 90.0712} C_DIS
LIN {X -1.9602,Y -8.2628,Z 28,A -3.1485,B 0,C 0,E1 0.1598,E2 90.0713} C_DIS
LIN {X -0.8412,Y -8.4495,Z 28,A -3.1155,B 0,C 0,E1 0.1598,E2 90.0713} C_DIS
LIN {X -0.8412,Y -8.4495,Z 28,A -3.1155,B 0,C 0,E1 0.1598,E2 90.0714} C_DIS
Enddeposition()
LIN {X 0.0007,Y -4.757,Z 29,A -2.9129,B 0,C 0,E1 0.1598,E2 90.0604} C_DIS
Startdeposition()
$VEL.CP = VEL_PRINT
LIN {X 0.0007,Y -4.757,Z 29,A -2.9186,B 0,C 0,E1 0.1598,E2 90.0661} C_DIS
LIN {X -0.6666,Y -4.7028,Z 29,A -2.9457,B 0,C 0,E1 0.1598,E2 90.071} C_DIS
LIN {X -1.3207,Y -4.5623,Z 29,A -2.9644,B 0,C 0,E1 0.1598,E2 90.0716} C_DIS
LIN {X -2.0351,Y -4.2906,Z 29,A -2.9791,B 0,C 0,E1 0.1598,E2 90.0716} C_DIS
LIN {X -2.5375,Y -4.0141,Z 29,A -2.9858,B 0,C 0,E1 0.1598,E2 90.0716} C_DIS
LIN {X -3.0035,Y -3.6798,Z 29,A -2.9888,B 0,C 0,E1 0.1598,E2 90.0716} C_DIS
LIN {X -3.5541,Y -3.1495,Z 29,A -2.9864,B 0,C 0,E1 0.1598,E2 90.0714} C_DIS
LIN {X -3.9083,Y -2.6986,Z 29,A -2.9803,B 0,C 0,E1 0.1598,E2 90.0714} C_DIS
LIN {X -4.2055,Y -2.2079,Z 29,A -2.9705,B 0,C 0,E1 0.1598,E2 90.0714} C_DIS
LIN {X -4.5041,Y -1.5044,Z 29,A -2.9516,B 0,C 0,E1 0.1598,E2 90.0714} C_DIS
LIN {X -4.6878,Y -0.7626,Z 29,A -2.9269,B 0,C 0,E1 0.1598,E2 90.0714} C_DIS
LIN {X -4.75,Y -0.0008,Z 29,A -2.897,B 0,C 0,E1 0.1598,E2 90.0714} C_DIS
LIN {X -4.6878,Y 0.761,Z 29,A -2.8625,B 0,C 0,E1 0.1598,E2 90.0714} C_DIS
LIN {X -4.5051,Y 1.5031,Z 29,A -2.8244,B 0,C 0,E1 0.1598,E2 90.0715} C_DIS
LIN {X -4.2071,Y 2.2071,Z 29,A -2.7837,B 0,C 0,E1 0.1598,E2 90.0716} C_DIS
LIN {X -3.7979,Y 2.8528,Z 29,A -2.7413,B 0,C 0,E1 0.1598,E2 90.0717} C_DIS
LIN {X -3.2906,Y 3.4246,Z 29,A -2.6985,B 0,C 0,E1 0.1598,E2 90.0718} C_DIS
LIN {X -2.6987,Y 3.9083,Z 29,A -2.6563,B 0,C 0,E1 0.1598,E2 90.0719} C_DIS
LIN {X -2.208,Y 4.2054,Z 29,A -2.6257,B 0,C 0,E1 0.1598,E2 90.072} C_DIS
LIN {X -1.5045,Y 4.5041,Z 29,A -2.5872,B 0,C 0,E1 0.1598,E2 90.072} C_DIS
LIN {X -0.9509,Y 4.6537,Z 29,A -2.5604,B 0,C 0,E1 0.1598,E2 90.0721} C_DIS
LIN {X -0.1922,Y 4.7468,Z 29,A -2.5285,B 0,C 0,E1 0.1598,E2 90.0721} C_DIS
LIN {X 0.5717,Y 4.7151,Z 29,A -2.5017,B 0,C 0,E1 0.1598,E2 90.0722} C_DIS
LIN {X 1.3209,Y 4.5633,Z 29,A -2.4805,B 0,C 0,E1 0.1598,E2 90.0722} C_DIS
LIN {X 2.0355,Y 4.2918,Z 29,A -2.4657,B 0,C 0,E1 0.1598,E2 90.0722} C_DIS
LIN {X 2.6978,Y 3.9097,Z 29,A -2.4574,B 0,C 0,E1 0.1598,E2 90.0722} C_DIS
LIN {X 3.2903,Y 3.4266,Z 29,A -2.456,B 0,C 0,E1 0.1598,E2 90.0722} C_DIS
LIN {X 3.7985,Y 2.8553,Z 29,A -2.4615,B 0,C 0,E1 0.1598,E2 90.0721} C_DIS
LIN {X 4.2061,Y 2.2082,Z 29,A -2.474,B 0,C 0,E1 0.1598,E2 90.0721} C_DIS
LIN {X 4.5045,Y 1.5045,Z 29,A -2.4928,B 0,C 0,E1 0.1598,E2 90.072} C_DIS
LIN {X 4.6537,Y 0.9508,Z 29,A -2.511,B 0,C 0,E1 0.1598,E2 90.072} C_DIS
LIN {X 4.7442,Y 0.1918,Z 29,A -2.5397,B 0,C 0,E1 0.1598,E2 90.0719} C_DIS
LIN {X 4.734,Y -0.3814,Z 29,A -2.5645,B 0,C 0,E1 0.1598,E2 90.0719} C_DIS
LIN {X 4.6116,Y -1.1359,Z 29,A -2.6011,B 0,C 0,E1 0.1598,E2 90.0718} C_DIS
LIN {X 4.3699,Y -1.8611,Z 29,A -2.6408,B 0,C 0,E1 0.1598,E2 90.0718} C_DIS
LIN {X 4.0154,Y -2.5383,Z 29,A -2.6827,B 0,C 0,E1 0.1598,E2 90.0718} C_DIS
LIN {X 3.5563,Y -3.1497,Z 29,A -2.7256,B 0,C 0,E1 0.1598,E2 90.0718} C_DIS
LIN {X 3.0055,Y -3.6801,Z 29,A -2.7684,B 0,C 0,E1 0.1598,E2 90.0718} C_DIS
LIN {X 2.3765,Y -4.115,Z 29,A -2.81,B 0,C 0,E1 0.1598,E2 90.0718} C_DIS
LIN {X 1.5952,Y -4.4741,Z 29,A -2.854,B 0,C 0,E1 0.1598,E2 90.0718} C_DIS
LIN {X 0.9508,Y -4.6538,Z 29,A -2.8853,B 0,C 0,E1 0.1598,E2 90.0718} C_DIS
LIN {X 0.192,Y -4.7489,Z 29,A -2.9172,B 0,C 0,E1 0.1598,E2 90.0717} C_DIS
LIN {X 0.192,Y -4.7489,Z 29,A -2.9172,B 0,C 0,E1 0.1598,E2 90.0717} C_DIS
Enddeposition()
LIN {X -0.0133,Y -5.6862,Z 29,A -2.9635,B 0,C 0,E1 0.1598,E2 90.0705} C_DIS
Startdeposition()
$VEL.CP = VEL_PRINT
LIN {X 0.6191,Y -5.6481,Z 29,A -2.9398,B 0,C 0,E1 0.1598,E2 90.0716} C_DIS
LIN {X 1.4488,Y -5.4937,Z 29,A -2.9029,B 0,C 0,E1 0.1598,E2 90.0716} C_DIS
LIN {X 2.2472,Y -5.2194,Z 29,A -2.8619,B 0,C 0,E1 0.1598,E2 90.0717} C_DIS
LIN {X 2.9952,Y -4.8282,Z 29,A -2.8178,B 0,C 0,E1 0.1598,E2 90.0717} C_DIS
LIN {X 3.6773,Y -4.3311,Z 29,A -2.7715,B 0,C 0,E1 0.1598,E2 90.0717} C_DIS
LIN {X 4.2791,Y -3.7391,Z 29,A -2.7242,B 0,C 0,E1 0.1598,E2 90.0717} C_DIS
LIN {X 4.7856,Y -3.0637,Z 29,A -2.6768,B 0,C 0,E1 0.1598,E2 90.0717} C_DIS
LIN {X 5.1869,Y -2.3211,Z 29,A -2.6304,B 0,C 0,E1 0.1598,E2 90.0717} C_DIS
LIN {X 5.4728,Y -1.5268,Z 29,A -2.586,B 0,C 0,E1 0.1598,E2 90.0717} C_DIS
LIN {X 5.6386,Y -0.6992,Z 29,A -2.5447,B 0,C 0,E1 0.1598,E2 90.0718} C_DIS
LIN {X 5.6813,Y 0.1438,Z 29,A -2.5072,B 0,C 0,E1 0.1598,E2 90.0718} C_DIS
LIN {X 5.5992,Y 0.9842,Z 29,A -2.4745,B 0,C 0,E1 0.1598,E2 90.0718} C_DIS
LIN {X 5.3921,Y 1.803,Z 29,A -2.4473,B 0,C 0,E1 0.1598,E2 90.0719} C_DIS
LIN {X 5.0653,Y 2.5818,Z 29,A -2.4263,B 0,C 0,E1 0.1598,E2 90.0719} C_DIS
LIN {X 4.6248,Y 3.3022,Z 29,A -2.4119,B 0,C 0,E1 0.1598,E2 90.072} C_DIS
LIN {X 4.085,Y 3.9514,Z 29,A -2.4043,B 0,C 0,E1 0.1598,E2 90.0721} C_DIS
LIN {X 3.4544,Y 4.5128,Z 29,A -2.4038,B 0,C 0,E1 0.1598,E2 90.0721} C_DIS
LIN {X 2.748,Y 4.9753,Z 29,A -2.4103,B 0,C 0,E1 0.1598,E2 90.0722} C_DIS
LIN {X 1.9809,Y 5.3283,Z 29,A -2.4236,B 0,C 0,E1 0.1598,E2 90.0722} C_DIS
LIN {X 1.1698,Y 5.5633,Z 29,A -2.4436,B 0,C 0,E1 0.1598,E2 90.0722} C_DIS
LIN {X 0.3328,Y 5.675,Z 29,A -2.4698,B 0,C 0,E1 0.1598,E2 90.0722} C_DIS
LIN {X -0.5116,Y 5.6623,Z 29,A -2.5015,B 0,C 0,E1 0.1598,E2 90.0722} C_DIS
LIN {X -1.345,Y 5.5247,Z 29,A -2.538,B 0,C 0,E1 0.1598,E2 90.0722} C_DIS
LIN {X -2.106,Y 5.2868,Z 29,A -2.5761,B 0,C 0,E1 0.1598,E2 90.0721} C_DIS
LIN {X -3.0284,Y 4.811,Z 29,A -2.6302,B 0,C 0,E1 0.1598,E2 90.072} C_DIS
LIN {X -3.6969,Y 4.3187,Z 29,A -2.6756,B 0,C 0,E1 0.1598,E2 90.0719} C_DIS
LIN {X -4.2858,Y 3.7336,Z 29,A -2.722,B 0,C 0,E1 0.1598,E2 90.0718} C_DIS
LIN {X -4.7846,Y 3.0699,Z 29,A -2.7684,B 0,C 0,E1 0.1598,E2 90.0717} C_DIS
LIN {X -5.1807,Y 2.3403,Z 29,A -2.8137,B 0,C 0,E1 0.1598,E2 90.0715} C_DIS
LIN {X -5.5464,Y 1.2703,Z 29,A -2.8721,B 0,C 0,E1 0.1598,E2 90.0712} C_DIS
LIN {X -5.671,Y 0.4096,Z 29,A -2.9133,B 0,C 0,E1 0.1598,E2 90.0713} C_DIS
LIN {X -5.6783,Y -0.286,Z 29,A -2.943,B 0,C 0,E1 0.1598,E2 90.0713} C_DIS
LIN {X -5.601,Y -0.9774,Z 29,A -2.9694,B 0,C 0,E1 0.1598,E2 90.0713} C_DIS
LIN {X -5.4392,Y -1.6539,Z 29,A -2.9921,B 0,C 0,E1 0.1598,E2 90.0713} C_DIS
LIN {X -5.1971,Y -2.3061,Z 29,A -3.0108,B 0,C 0,E1 0.1598,E2 90.0713} C_DIS
LIN {X -4.875,Y -2.9226,Z 29,A -3.0251,B 0,C 0,E1 0.1598,E2 90.0713} C_DIS
LIN {X -4.2655,Y -3.7651,Z 29,A -3.0382,B 0,C 0,E1 0.1598,E2 90.0712} C_DIS
LIN {X -3.5966,Y -4.4018,Z 29,A -3.0407,B 0,C 0,E1 0.1598,E2 90.0713} C_DIS
LIN {X -2.995,Y -4.8304,Z 29,A -3.0369,B 0,C 0,E1 0.1598,E2 90.0714} C_DIS
LIN {X -2.3436,Y -5.1784,Z 29,A -3.0278,B 0,C 0,E1 0.1598,E2 90.0714} C_DIS
LIN {X -1.6525,Y -5.4394,Z 29,A -3.0135,B 0,C 0,E1 0.1598,E2 90.0715} C_DIS
LIN {X -0.9334,Y -5.609,Z 29,A -2.9944,B 0,C 0,E1 0.1598,E2 90.0715} C_DIS
LIN {X -0.0133,Y -5.6862,Z 29,A -2.9639,B 0,C 0,E1 0.1598,E2 90.0716} C_DIS
Enddeposition()
LIN {X -0.0133,Y -5.6862,Z 29,A -2.9639,B 0,C 0,E1 0.1598,E2 90.0716} C_DIS
Startdeposition()
$VEL.CP = VEL_PRINT
LIN {X -0.6208,Y -6.5907,Z 29,A -3.0242,B 0,C 0,E1 0.1598,E2 90.071} C_DIS
LIN {X -1.3808,Y -6.4718,Z 29,A -3.0475,B 0,C 0,E1 0.1598,E2 90.0715} C_DIS
LIN {X -2.1223,Y -6.2676,Z 29,A -3.0661,B 0,C 0,E1 0.1598,E2 90.0715} C_DIS
LIN {X -2.8355,Y -5.9798,Z 29,A -3.08,B 0,C 0,E1 0.1598,E2 90.0715} C_DIS
LIN {X -3.5119,Y -5.6133,Z 29,A -3.0893,B 0,C 0,E1 0.1598,E2 90.0714} C_DIS
LIN {X -4.1379,Y -5.1663,Z 29,A -3.0933,B 0,C 0,E1 0.1598,E2 90.0714} C_DIS
LIN {X -4.7092,Y -4.651,Z 29,A -3.0924,B 0,C 0,E1 0.1598,E2 90.0714} C_DIS
LIN {X -5.2165,Y -4.0727,Z 29,A -3.0865,B 0,C 0,E1 0.1598,E2 90.0713} C_DIS
LIN {X -5.6539,Y -3.44,Z 29,A -3.0757,B 0,C 0,E1 0.1598,E2 90.0713} C_DIS
LIN {X -6.0146,Y -2.7607,Z 29,A -3.0602,B 0,C 0,E1 0.1598,E2 90.0713} C_DIS
LIN {X -6.2939,Y -2.0441,Z 29,A -3.0401,B 0,C 0,E1 0.1598,E2 90.0713} C_DIS
LIN {X -6.4899,Y -1.3003,Z 29,A -3.0159,B 0,C 0,E1 0.1598,E2 90.0713} C_DIS
LIN {X -6.5981,Y -0.5386,Z 29,A -2.9877,B 0,C 0,E1 0.1598,E2 90.0713} C_DIS
LIN {X -6.6161,Y 0.2303,Z 29,A -2.9558,B 0,C 0,E1 0.1598,E2 90.0713} C_DIS
LIN {X -6.5446,Y 0.9964,Z 29,A -2.9209,B 0,C 0,E1 0.1598,E2 90.0713} C_DIS
LIN {X -6.3856,Y 1.749,Z 29,A -2.8832,B 0,C 0,E1 0.1598,E2 90.0714} C_DIS
LIN {X -6.1392,Y 2.4777,Z 29,A -2.8434,B 0,C 0,E1 0.1598,E2 90.0715} C_DIS
LIN {X -5.8115,Y 3.1737,Z 29,A -2.802,B 0,C 0,E1 0.1598,E2 90.0715} C_DIS
LIN {X -5.4017,Y 3.8247,Z 29,A -2.7594,B 0,C 0,E1 0.1598,E2 90.0717} C_DIS
LIN {X -4.9223,Y 4.4264,Z 29,A -2.7163,B 0,C 0,E1 0.1598,E2 90.0717} C_DIS
LIN {X -4.3747,Y 4.9668,Z 29,A -2.6734,B 0,C 0,E1 0.1598,E2 90.0719} C_DIS
LIN {X -3.7684,Y 5.4402,Z 29,A -2.631,B 0,C 0,E1 0.1598,E2 90.0719} C_DIS
LIN {X -3.112,Y 5.8414,Z 29,A -2.5899,B 0,C 0,E1 0.1598,E2 90.072} C_DIS
LIN {X -2.4136,Y 6.1638,Z 29,A -2.5505,B 0,C 0,E1 0.1598,E2 90.0721} C_DIS
LIN {X -1.6817,Y 6.4008,Z 29,A -2.5135,B 0,C 0,E1 0.1598,E2 90.0721} C_DIS
LIN {X -0.9278,Y 6.5531,Z 29,A -2.4793,B 0,C 0,E1 0.1598,E2 90.0723} C_DIS
LIN {X -0.1612,Y 6.6175,Z 29,A -2.4483,B 0,C 0,E1 0.1598,E2 90.0723} C_DIS
LIN {X 0.6075,Y 6.5896,Z 29,A -2.4211,B 0,C 0,E1 0.1598,E2 90.0723} C_DIS
LIN {X 1.3683,Y 6.4761,Z 29,A -2.3978,B 0,C 0,E1 0.1598,E2 90.0723} C_DIS
LIN {X 2.1107,Y 6.2747,Z 29,A -2.379,B 0,C 0,E1 0.1598,E2 90.0723} C_DIS
LIN {X 3.124,Y 5.8403,Z 29,A -2.3599,B 0,C 0,E1 0.1598,E2 90.0723} C_DIS
LIN {X 3.9436,Y 5.3171,Z 29,A -2.3518,B 0,C 0,E1 0.1598,E2 90.0723} C_DIS
LIN {X 4.5395,Y 4.8172,Z 29,A -2.3511,B 0,C 0,E1 0.1598,E2 90.0723} C_DIS
LIN {X 5.0729,Y 4.2511,Z 29,A -2.3554,B 0,C 0,E1 0.1598,E2 90.0723} C_DIS
LIN {X 5.5363,Y 3.6267,Z 29,A -2.3648,B 0,C 0,E1 0.1598,E2 90.0722} C_DIS
LIN {X 5.9232,Y 2.952,Z 29,A -2.3792,B 0,C 0,E1 0.1598,E2 90.0722} C_DIS
LIN {X 6.23,Y 2.2372,Z 29,A -2.3983,B 0,C 0,E1 0.1598,E2 90.0721} C_DIS
LIN {X 6.4494,Y 1.491,Z 29,A -2.4219,B 0,C 0,E1 0.1598,E2 90.0721} C_DIS
LIN {X 6.5775,Y 0.7239,Z 29,A -2.4498,B 0,C 0,E1 0.1598,E2 90.072} C_DIS
LIN {X 6.6174,Y -0.0526,Z 29,A -2.4814,B 0,C 0,E1 0.1598,E2 90.072} C_DIS
LIN {X 6.568,Y -0.8287,Z 29,A -2.5163,B 0,C 0,E1 0.1598,E2 90.0719} C_DIS
LIN {X 6.4253,Y -1.5935,Z 29,A -2.5541,B 0,C 0,E1 0.1598,E2 90.0719} C_DIS
LIN {X 6.1951,Y -2.3364,Z 29,A -2.5942,B 0,C 0,E1 0.1598,E2 90.0719} C_DIS
LIN {X 5.8775,Y -3.0464,Z 29,A -2.6361,B 0,C 0,E1 0.1598,E2 90.0718} C_DIS
LIN {X 5.4804,Y -3.7151,Z 29,A -2.6792,B 0,C 0,E1 0.1598,E2 90.0718} C_DIS
LIN {X 5.0044,Y -4.3303,Z 29,A -2.7229,B 0,C 0,E1 0.1598,E2 90.0718} C_DIS
LIN {X 4.4626,Y -4.8882,Z 29,A -2.7665,B 0,C 0,E1 0.1598,E2 90.0718} C_DIS
LIN {X 3.7011,Y -5.4927,Z 29,A -2.8202,B 0,C 0,E1 0.1598,E2 90.0716} C_DIS
LIN {X 2.7577,Y -6.0176,Z 29,A -2.8772,B 0,C 0,E1 0.1598,E2 90.0716} C_DIS
LIN {X 2.0403,Y -6.2971,Z 29,A -2.9155,B 0,C 0,E1 0.1598,E2 90.0716} C_DIS
LIN {X 1.2949,Y -6.4895,Z 29,A -2.951,B 0,C 0,E1 0.1598,E2 90.0716} C_DIS
LIN {X 0.5327,Y -6.5966,Z 29,A -2.9835,B 0,C 0,E1 0.1598,E2 90.0716} C_DIS
LIN {X 0.5327,Y -6.5966,Z 29,A -2.9835,B 0,C 0,E1 0.1598,E2 90.0716} C_DIS
Enddeposition()
LIN {X -0.0423,Y -7.5529,Z 29,A -3.0442,B 0,C 0,E1 0.1598,E2 90.0703} C_DIS
Startdeposition()
$VEL.CP = VEL_PRINT
LIN {X 0.8187,Y -7.5124,Z 29,A -3.0121,B 0,C 0,E1 0.1598,E2 90.0715} C_DIS
LIN {X 2.0741,Y -7.2685,Z 29,A -2.9557,B 0,C 0,E1 0.1598,E2 90.0716} C_DIS
LIN {X 3.0258,Y -6.9247,Z 29,A -2.9061,B 0,C 0,E1 0.1598,E2 90.0716} C_DIS
LIN {X 3.926,Y -6.4567,Z 29,A -2.8532,B 0,C 0,E1 0.1598,E2 90.0716} C_DIS
LIN {X 4.768,Y -5.8568,Z 29,A -2.7967,B 0,C 0,E1 0.1598,E2 90.0716} C_DIS
LIN {X 5.5262,Y -5.1541,Z 29,A -2.7388,B 0,C 0,E1 0.1598,E2 90.0716} C_DIS
LIN {X 6.1549,Y -4.385,Z 29,A -2.683,B 0,C 0,E1 0.1598,E2 90.0716} C_DIS
LIN {X 6.8051,Y -3.2851,Z 29,A -2.6119,B 0,C 0,E1 0.1598,E2 90.0716} C_DIS
LIN {X 7.2027,Y -2.2755,Z 29,A -2.5544,B 0,C 0,E1 0.1598,E2 90.0716} C_DIS
LIN {X 7.4151,Y -1.4338,Z 29,A -2.5108,B 0,C 0,E1 0.1598,E2 90.0718} C_DIS
LIN {X 7.5307,Y -0.5735,Z 29,A -2.4699,B 0,C 0,E1 0.1598,E2 90.0718} C_DIS
LIN {X 7.5329,Y 0.6101,Z 29,A -2.4191,B 0,C 0,E1 0.1598,E2 90.0716} C_DIS
LIN {X 7.3912,Y 1.5733,Z 29,A -2.3836,B 0,C 0,E1 0.1598,E2 90.0719} C_DIS
LIN {X 7.1087,Y 2.5633,Z 29,A -2.3518,B 0,C 0,E1 0.1598,E2 90.0719} C_DIS
LIN {X 6.7016,Y 3.4831,Z 29,A -2.3277,B 0,C 0,E1 0.1598,E2 90.072} C_DIS
LIN {X 6.2936,Y 4.1767,Z 29,A -2.3135,B 0,C 0,E1 0.1598,E2 90.0722} C_DIS
LIN {X 5.8133,Y 4.8224,Z 29,A -2.3038,B 0,C 0,E1 0.1598,E2 90.0722} C_DIS
LIN {X 5.2673,Y 5.4137,Z 29,A -2.2988,B 0,C 0,E1 0.1598,E2 90.0722} C_DIS
LIN {X 4.4116,Y 6.1366,Z 29,A -2.2996,B 0,C 0,E1 0.1598,E2 90.0722} C_DIS
LIN {X 3.4731,Y 6.7065,Z 29,A -2.3101,B 0,C 0,E1 0.1598,E2 90.0722} C_DIS
LIN {X 2.4662,Y 7.1444,Z 29,A -2.3288,B 0,C 0,E1 0.1598,E2 90.0723} C_DIS
LIN {X 1.2648,Y 7.4474,Z 29,A -2.3604,B 0,C 0,E1 0.1598,E2 90.0723} C_DIS
LIN {X 0.5221,Y 7.5389,Z 29,A -2.384,B 0,C 0,E1 0.1598,E2 90.0723} C_DIS
LIN {X -0.4709,Y 7.5423,Z 29,A -2.4205,B 0,C 0,E1 0.1598,E2 90.0723} C_DIS
LIN {X -1.4052,Y 7.4264,Z 29,A -2.4599,B 0,C 0,E1 0.1598,E2 90.0723} C_DIS
LIN {X -2.726,Y 7.0489,Z 29,A -2.5245,B 0,C 0,E1 0.1598,E2 90.0721} C_DIS
LIN {X -3.5431,Y 6.6753,Z 29,A -2.5704,B 0,C 0,E1 0.1598,E2 90.0721} C_DIS
LIN {X -4.2649,Y 6.2367,Z 29,A -2.6156,B 0,C 0,E1 0.1598,E2 90.072} C_DIS
LIN {X -5.06,Y 5.6151,Z 29,A -2.671,B 0,C 0,E1 0.1598,E2 90.0718} C_DIS
LIN {X -5.7516,Y 4.8971,Z 29,A -2.7268,B 0,C 0,E1 0.1598,E2 90.0718} C_DIS
LIN {X -6.4541,Y 3.9302,Z 29,A -2.7933,B 0,C 0,E1 0.1598,E2 90.0714} C_DIS
LIN {X -7.0526,Y 2.7159,Z 29,A -2.8663,B 0,C 0,E1 0.1598,E2 90.071} C_DIS
LIN {X -7.3858,Y 1.599,Z 29,A -2.9257,B 0,C 0,E1 0.1598,E2 90.071} C_DIS
LIN {X -7.5396,Y 0.5111,Z 29,A -2.9774,B 0,C 0,E1 0.1598,E2 90.071} C_DIS
LIN {X -7.539,Y -0.5199,Z 29,A -3.0209,B 0,C 0,E1 0.1598,E2 90.071} C_DIS
LIN {X -7.4085,Y -1.4906,Z 29,A -3.0572,B 0,C 0,E1 0.1598,E2 90.071} C_DIS
LIN {X -7.0293,Y -2.7788,Z 29,A -3.0974,B 0,C 0,E1 0.1598,E2 90.0707} C_DIS
LIN {X -6.5198,Y -3.8139,Z 29,A -3.1226,B 0,C 0,E1 0.1598,E2 90.0707} C_DIS
LIN {X -6.0535,Y -4.5163,Z 29,A -3.1355,B 0,C 0,E1 0.1598,E2 90.0711} C_DIS
LIN {X -5.5128,Y -5.1634,Z 29,A -3.1431,B 0,C 0,E1 0.1598,E2 90.0711} C_DIS
LIN {X -4.7438,Y -5.8842,Z 29,A -3.1453,B 0,C 0,E1 0.1598,E2 90.0711} C_DIS
LIN {X -3.7239,Y -6.5716,Z 29,A -3.1371,B 0,C 0,E1 0.1598,E2 90.0711} C_DIS
LIN {X -3.0328,Y -6.9217,Z 29,A -3.1267,B 0,C 0,E1 0.1598,E2 90.0713} C_DIS
LIN {X -1.7494,Y -7.3531,Z 29,A -3.098,B 0,C 0,E1 0.1598,E2 90.0713} C_DIS
LIN {X -0.7943,Y -7.5152,Z 29,A -3.0699,B 0,C 0,E1 0.1598,E2 90.0715} C_DIS
LIN {X -0.0423,Y -7.5529,Z 29,A -3.044,B 0,C 0,E1 0.1598,E2 90.0715} C_DIS
Enddeposition()
LIN {X -0.0423,Y -7.5529,Z 29,A -3.044,B 0,C 0,E1 0.1598,E2 90.0715} C_DIS
Startdeposition()
$VEL.CP = VEL_PRINT
LIN {X -0.8417,Y -8.4494,Z 29,A -3.111,B 0,C 0,E1 0.1598,E2 90.0709} C_DIS
LIN {X -2.0289,Y -8.2451,Z 29,A -3.1463,B 0,C 0,E1 0.1598,E2 90.0713} C_DIS
LIN {X -3.0371,Y -7.9238,Z 29,A -3.1697,B 0,C 0,E1 0.1598,E2 90.0713} C_DIS
LIN {X -3.8114,Y -7.5817,Z 29,A -3.1835,B 0,C 0,E1 0.1598,E2 90.0713} C_DIS
LIN {X -4.5477,Y -7.1642,Z 29,A -3.1928,B 0,C 0,E1 0.1598,E2 90.0713} C_DIS
LIN {X -5.2389,Y -6.6755,Z 29,A -3.1974,B 0,C 0,E1 0.1598,E2 90.0712} C_DIS
LIN {X -5.8781,Y -6.1205,Z 29,A -3.1974,B 0,C 0,E1 0.1598,E2 90.0712} C_DIS
LIN {X -6.4588,Y -5.5047,Z 29,A -3.1925,B 0,C 0,E1 0.1598,E2 90.0712} C_DIS
LIN {X -6.9754,Y -4.8341,Z 29,A -3.1831,B 0,C 0,E1 0.1598,E2 90.0711} C_DIS
LIN {X -7.4226,Y -4.1154,Z 29,A -3.1691,B 0,C 0,E1 0.1598,E2 90.0711} C_DIS
LIN {X -7.7957,Y -3.3556,Z 29,A -3.1506,B 0,C 0,E1 0.1598,E2 90.0711} C_DIS
LIN {X -8.0911,Y -2.5623,Z 29,A -3.1279,B 0,C 0,E1 0.1598,E2 90.0711} C_DIS
LIN {X -8.367,Y -1.4458,Z 29,A -3.0907,B 0,C 0,E1 0.1598,E2 90.0709} C_DIS
LIN {X -8.4808,Y -0.43,Z 29,A -3.0519,B 0,C 0,E1 0.1598,E2 90.0709} C_DIS
LIN {X -8.4718,Y 0.5635,Z 29,A -3.0098,B 0,C 0,E1 0.1598,E2 90.071} C_DIS
LIN {X -8.2925,Y 1.8126,Z 29,A -2.9502,B 0,C 0,E1 0.1598,E2 90.0708} C_DIS
LIN {X -8.0728,Y 2.6313,Z 29,A -2.9078,B 0,C 0,E1 0.1598,E2 90.0711} C_DIS
LIN {X -7.703,Y 3.5618,Z 29,A -2.8551,B 0,C 0,E1 0.1598,E2 90.0714} C_DIS
LIN {X -7.3336,Y 4.2727,Z 29,A -2.8116,B 0,C 0,E1 0.1598,E2 90.0716} C_DIS
LIN {X -6.7818,Y 5.1083,Z 29,A -2.7559,B 0,C 0,E1 0.1598,E2 90.0715} C_DIS
LIN {X -6.0408,Y 5.9681,Z 29,A -2.6923,B 0,C 0,E1 0.1598,E2 90.0716} C_DIS
LIN {X -5.1168,Y 6.773,Z 29,A -2.6243,B 0,C 0,E1 0.1598,E2 90.0717} C_DIS
LIN {X -4.4156,Y 7.2502,Z 29,A -2.5785,B 0,C 0,E1 0.1598,E2 90.072} C_DIS
LIN {X -3.6701,Y 7.6548,Z 29,A -2.5339,B 0,C 0,E1 0.1598,E2 90.0721} C_DIS
LIN {X -2.8879,Y 7.9827,Z 29,A -2.4912,B 0,C 0,E1 0.1598,E2 90.0721} C_DIS
LIN {X -2.0769,Y 8.2308,Z 29,A -2.4508,B 0,C 0,E1 0.1598,E2 90.0723} C_DIS
LIN {X -0.8638,Y 8.4469,Z 29,A -2.3969,B 0,C 0,E1 0.1598,E2 90.0723} C_DIS
LIN {X 0.1855,Y 8.4885,Z 29,A -2.3564,B 0,C 0,E1 0.1598,E2 90.0724} C_DIS
LIN {X 1.2708,Y 8.3951,Z 29,A -2.3202,B 0,C 0,E1 0.1598,E2 90.0724} C_DIS
LIN {X 2.2711,Y 8.182,Z 29,A -2.2923,B 0,C 0,E1 0.1598,E2 90.0724} C_DIS
LIN {X 3.2716,Y 7.8332,Z 29,A -2.2701,B 0,C 0,E1 0.1598,E2 90.0724} C_DIS
LIN {X 4.0364,Y 7.4678,Z 29,A -2.2574,B 0,C 0,E1 0.1598,E2 90.0724} C_DIS
LIN {X 5.0248,Y 6.8459,Z 29,A -2.2471,B 0,C 0,E1 0.1598,E2 90.0724} C_DIS
LIN {X 5.9377,Y 6.0653,Z 29,A -2.2464,B 0,C 0,E1 0.1598,E2 90.0722} C_DIS
LIN {X 6.5136,Y 5.4427,Z 29,A -2.2518,B 0,C 0,E1 0.1598,E2 90.0723} C_DIS
LIN {X 7.0245,Y 4.7658,Z 29,A -2.2617,B 0,C 0,E1 0.1598,E2 90.0723} C_DIS
LIN {X 7.4653,Y 4.0412,Z 29,A -2.2762,B 0,C 0,E1 0.1598,E2 90.0723} C_DIS
LIN {X 7.9133,Y 3.0805,Z 29,A -2.3003,B 0,C 0,E1 0.1598,E2 90.0719} C_DIS
LIN {X 8.2304,Y 2.0686,Z 29,A -2.3317,B 0,C 0,E1 0.1598,E2 90.0719} C_DIS
LIN {X 8.4295,Y 1.0172,Z 29,A -2.3691,B 0,C 0,E1 0.1598,E2 90.0717} C_DIS
LIN {X 8.4913,Y 0.0632,Z 29,A -2.4075,B 0,C 0,E1 0.1598,E2 90.0717} C_DIS
LIN {X 8.4404,Y -0.9216,Z 29,A -2.4513,B 0,C 0,E1 0.1598,E2 90.0717} C_DIS
LIN {X 8.2844,Y -1.8629,Z 29,A -2.4972,B 0,C 0,E1 0.1598,E2 90.0717} C_DIS
LIN {X 7.9358,Y -3.0191,Z 29,A -2.5591,B 0,C 0,E1 0.1598,E2 90.0714} C_DIS
LIN {X 7.3817,Y -4.196,Z 29,A -2.6296,B 0,C 0,E1 0.1598,E2 90.0714} C_DIS
LIN {X 6.7565,Y -5.1412,Z 29,A -2.6931,B 0,C 0,E1 0.1598,E2 90.0715} C_DIS
LIN {X 6.0618,Y -5.9411,Z 29,A -2.7528,B 0,C 0,E1 0.1598,E2 90.0715} C_DIS
LIN {X 5.4393,Y -6.5163,Z 29,A -2.8003,B 0,C 0,E1 0.1598,E2 90.0717} C_DIS
LIN {X 4.7625,Y -7.0267,Z 29,A -2.8469,B 0,C 0,E1 0.1598,E2 90.0717} C_DIS
LIN {X 4.0382,Y -7.4669,Z 29,A -2.8922,B 0,C 0,E1 0.1598,E2 90.0717} C_DIS
LIN {X 3.2734,Y -7.8322,Z 29,A -2.9358,B 0,C 0,E1 0.1598,E2 90.0717} C_DIS
LIN {X 2.4761,Y -8.1197,Z 29,A -2.9773,B 0,C 0,E1 0.1598,E2 90.0716} C_DIS
LIN {X 1.6539,Y -8.3257,Z 29,A -3.0162,B 0,C 0,E1 0.1598,E2 90.0716} C_DIS
LIN {X 0.4294,Y -8.4808,Z 29,A -3.0677,B 0,C 0,E1 0.1598,E2 90.0715} C_DIS
LIN {X 0.4294,Y -8.4808,Z 29,A -3.0677,B 0,C 0,E1 0.1598,E2 90.0715} C_DIS
Enddeposition()
LIN {X 0.0007,Y -4.7568,Z 30,A -2.9103,B 0,C 0,E1 0.1598,E2 90.0604} C_DIS
Startdeposition()
$VEL.CP = VEL_PRINT
LIN {X 0.0007,Y -4.7568,Z 30,A -2.916,B 0,C 0,E1 0.1598,E2 90.0661} C_DIS
LIN {X 0.9139,Y -4.6625,Z 30,A -2.8834,B 0,C 0,E1 0.1598,E2 90.0711} C_DIS
LIN {X 1.6209,Y -4.4642,Z 30,A -2.8496,B 0,C 0,E1 0.1598,E2 90.0717} C_DIS
LIN {X 2.2895,Y -4.1609,Z 30,A -2.8122,B 0,C 0,E1 0.1598,E2 90.0717} C_DIS
LIN {X 2.9046,Y -3.7594,Z 30,A -2.7725,B 0,C 0,E1 0.1598,E2 90.0717} C_DIS
LIN {X 3.3241,Y -3.4015,Z 30,A -2.7419,B 0,C 0,E1 0.1598,E2 90.0719} C_DIS
LIN {X 4.0018,Y -2.5583,Z 30,A -2.6808,B 0,C 0,E1 0.1598,E2 90.0716} C_DIS
LIN {X 4.3562,Y -1.8933,Z 30,A -2.6397,B 0,C 0,E1 0.1598,E2 90.0718} C_DIS
LIN {X 4.6004,Y -1.1803,Z 30,A -2.6003,B 0,C 0,E1 0.1598,E2 90.0718} C_DIS
LIN {X 4.7312,Y -0.4379,Z 30,A -2.5639,B 0,C 0,E1 0.1598,E2 90.0718} C_DIS
LIN {X 4.7315,Y 0.4096,Z 30,A -2.5277,B 0,C 0,E1 0.1598,E2 90.0718} C_DIS
LIN {X 4.6311,Y 1.0616,Z 30,A -2.5039,B 0,C 0,E1 0.1598,E2 90.072} C_DIS
LIN {X 4.406,Y 1.7812,Z 30,A -2.4815,B 0,C 0,E1 0.1598,E2 90.072} C_DIS
LIN {X 4.0667,Y 2.4544,Z 30,A -2.4655,B 0,C 0,E1 0.1598,E2 90.072} C_DIS
LIN {X 3.6261,Y 3.066,Z 30,A -2.4558,B 0,C 0,E1 0.1598,E2 90.072} C_DIS
LIN {X 3.0953,Y 3.6007,Z 30,A -2.4527,B 0,C 0,E1 0.1598,E2 90.0721} C_DIS
LIN {X 2.4874,Y 4.0459,Z 30,A -2.4562,B 0,C 0,E1 0.1598,E2 90.0721} C_DIS
LIN {X 1.8162,Y 4.3888,Z 30,A -2.4665,B 0,C 0,E1 0.1598,E2 90.0722} C_DIS
LIN {X 1.0989,Y 4.6197,Z 30,A -2.4831,B 0,C 0,E1 0.1598,E2 90.0722} C_DIS
LIN {X 0.3545,Y 4.736,Z 30,A -2.5057,B 0,C 0,E1 0.1598,E2 90.0722} C_DIS
LIN {X -0.399,Y 4.7326,Z 30,A -2.5336,B 0,C 0,E1 0.1598,E2 90.0722} C_DIS
LIN {X -1.1424,Y 4.6094,Z 30,A -2.5662,B 0,C 0,E1 0.1598,E2 90.0722} C_DIS
LIN {X -1.8576,Y 4.3717,Z 30,A -2.6026,B 0,C 0,E1 0.1598,E2 90.0721} C_DIS
LIN {X -2.5268,Y 4.0246,Z 30,A -2.642,B 0,C 0,E1 0.1598,E2 90.072} C_DIS
LIN {X -3.131,Y 3.5736,Z 30,A -2.6833,B 0,C 0,E1 0.1598,E2 90.0719} C_DIS
LIN {X -3.6564,Y 3.033,Z 30,A -2.7254,B 0,C 0,E1 0.1598,E2 90.0718} C_DIS
LIN {X -4.0887,Y 2.4156,Z 30,A -2.7674,B 0,C 0,E1 0.1598,E2 90.0717} C_DIS
LIN {X -4.4211,Y 1.7393,Z 30,A -2.8082,B 0,C 0,E1 0.1598,E2 90.0716} C_DIS
LIN {X -4.6414,Y 1.0182,Z 30,A -2.8468,B 0,C 0,E1 0.1598,E2 90.0716} C_DIS
LIN {X -4.7425,Y 0.2712,Z 30,A -2.882,B 0,C 0,E1 0.1598,E2 90.0714} C_DIS
LIN {X -4.7253,Y -0.4822,Z 30,A -2.9133,B 0,C 0,E1 0.1598,E2 90.0714} C_DIS
LIN {X -4.5903,Y -1.2237,Z 30,A -2.9397,B 0,C 0,E1 0.1598,E2 90.0714} C_DIS
LIN {X -4.3377,Y -1.9338,Z 30,A -2.9605,B 0,C 0,E1 0.1598,E2 90.0714} C_DIS
LIN {X -3.9766,Y -2.5951,Z 30,A -2.9752,B 0,C 0,E1 0.1598,E2 90.0714} C_DIS
LIN {X -3.5165,Y -3.1919,Z 30,A -2.9836,B 0,C 0,E1 0.1598,E2 90.0714} C_DIS
LIN {X -2.9674,Y -3.708,Z 30,A -2.9854,B 0,C 0,E1 0.1598,E2 90.0714} C_DIS
LIN {X -2.343,Y -4.1297,Z 30,A -2.9804,B 0,C 0,E1 0.1598,E2 90.0714} C_DIS
LIN {X -1.6607,Y -4.4492,Z 30,A -2.9689,B 0,C 0,E1 0.1598,E2 90.0716} C_DIS
LIN {X -0.9361,Y -4.6565,Z 30,A -2.9511,B 0,C 0,E1 0.1598,E2 90.0716} C_DIS
LIN {X -0.188,Y -4.7488,Z 30,A -2.9276,B 0,C 0,E1 0.1598,E2 90.0716} C_DIS
LIN {X -0.188,Y -4.7488,Z 30,A -2.9276,B 0,C 0,E1 0.1598,E2 90.0716} C_DIS
Enddeposition()
LIN {X -0.022,Y -5.6862,Z 30,A -2.9603,B 0,C 0,E1 0.1598,E2 90.0705} C_DIS
Startdeposition()
$VEL.CP = VEL_PRINT
LIN {X -1.0161,Y -5.5945,Z 30,A -2.9939,B 0,C 0,E1 0.1598,E2 90.0715} C_DIS
LIN {X -1.7896,Y -5.3947,Z 30,A -3.0139,B 0,C 0,E1 0.1598,E2 90.0715} C_DIS
LIN {X -2.5282,Y -5.091,Z 30,A -3.0281,B 0,C 0,E1 0.1598,E2 90.0715} C_DIS
LIN {X -3.2165,Y -4.6857,Z 30,A -3.0361,B 0,C 0,E1 0.1598,E2 90.0715} C_DIS
LIN {X -3.8408,Y -4.1878,Z 30,A -3.0379,B 0,C 0,E1 0.1598,E2 90.0714} C_DIS
LIN {X -4.5912,Y -3.3625,Z 30,A -3.0303,B 0,C 0,E1 0.1598,E2 90.0712} C_DIS
LIN {X -5.0446,Y -2.6199,Z 30,A -3.0156,B 0,C 0,E1 0.1598,E2 90.0712} C_DIS
LIN {X -5.3293,Y -1.9847,Z 30,A -2.9993,B 0,C 0,E1 0.1598,E2 90.0714} C_DIS
LIN {X -5.5311,Y -1.3185,Z 30,A -2.9785,B 0,C 0,E1 0.1598,E2 90.0714} C_DIS
LIN {X -5.6496,Y -0.6326,Z 30,A -2.9538,B 0,C 0,E1 0.1598,E2 90.0714} C_DIS
LIN {X -5.6853,Y 0.0624,Z 30,A -2.9257,B 0,C 0,E1 0.1598,E2 90.0714} C_DIS
LIN {X -5.636,Y 0.7568,Z 30,A -2.8946,B 0,C 0,E1 0.1598,E2 90.0714} C_DIS
LIN {X -5.4105,Y 1.7609,Z 30,A -2.8436,B 0,C 0,E1 0.1598,E2 90.0713} C_DIS
LIN {X -5.016,Y 2.6739,Z 30,A -2.7906,B 0,C 0,E1 0.1598,E2 90.0715} C_DIS
LIN {X -4.594,Y 3.3484,Z 30,A -2.7467,B 0,C 0,E1 0.1598,E2 90.0717} C_DIS
LIN {X -4.0818,Y 3.9573,Z 30,A -2.7021,B 0,C 0,E1 0.1598,E2 90.0717} C_DIS
LIN {X -3.4892,Y 4.4882,Z 30,A -2.6579,B 0,C 0,E1 0.1598,E2 90.0719} C_DIS
LIN {X -2.6564,Y 5.0319,Z 30,A -2.6041,B 0,C 0,E1 0.1598,E2 90.0719} C_DIS
LIN {X -1.4959,Y 5.4897,Z 30,A -2.5421,B 0,C 0,E1 0.1598,E2 90.0721} C_DIS
LIN {X -0.8765,Y 5.6165,Z 30,A -2.5139,B 0,C 0,E1 0.1598,E2 90.0722} C_DIS
LIN {X -0.0368,Y 5.6831,Z 30,A -2.4801,B 0,C 0,E1 0.1598,E2 90.0722} C_DIS
LIN {X 0.8033,Y 5.6257,Z 30,A -2.4516,B 0,C 0,E1 0.1598,E2 90.0722} C_DIS
LIN {X 1.6258,Y 5.4449,Z 30,A -2.4289,B 0,C 0,E1 0.1598,E2 90.0723} C_DIS
Enddeposition()
END
